C09142=1197.149,49.616,-46.613,-179.290,5.761,148.809
C09143=1197.154,49.367,-46.596,-179.293,5.760,148.810
C09144=1197.159,49.117,-46.581,-179.295,5.760,148.811
C09145=1197.164,48.868,-46.565,-179.298,5.759,148.811
C09146=1197.169,48.618,-46.548,-179.300,5.759,148.812
C09147=1197.174,48.369,-46.533,-179.303,5.758,148.812
C09148=1197.179,48.120,-46.516,-179.306,5.757,148.813
C09149=1197.184,47.870,-46.501,-179.308,5.756,148.813
C09150=1197.189,47.621,-46.484,-179.311,5.755,148.814
C09151=1197.194,47.371,-46.468,-179.313,5.755,148.815
C09152=1197.199,47.122,-46.453,-179.316,5.754,148.815
C09153=1197.204,46.872,-46.436,-179.318,5.753,148.816
C09154=1197.209,46.623,-46.421,-179.321,5.753,148.817
C09155=1197.213,46.373,-46.405,-179.323,5.752,148.817
C09156=1197.218,46.124,-46.389,-179.326,5.751,148.818
C09157=1197.223,45.874,-46.373,-179.329,5.750,148.818
C09158=1197.229,45.625,-46.357,-179.331,5.749,148.819
C09159=1197.234,45.376,-46.341,-179.334,5.749,148.820
C09160=1197.238,45.126,-46.325,-179.336,5.748,148.820
C09161=1197.244,44.877,-46.309,-179.339,5.748,148.821
C09162=1197.249,44.628,-46.293,-179.341,5.747,148.821
C09163=1197.253,44.378,-46.278,-179.344,5.746,148.822
C09164=1197.258,44.129,-46.262,-179.346,5.746,148.823
C09165=1197.263,43.879,-46.246,-179.349,5.744,148.823
C09166=1197.268,43.630,-46.230,-179.352,5.744,148.824
C09167=1197.274,43.380,-46.214,-179.354,5.743,148.824
C09168=1197.278,43.130,-46.198,-179.357,5.742,148.825
C09169=1197.284,42.881,-46.182,-179.360,5.742,148.826
C09170=1197.288,42.632,-46.167,-179.362,5.741,148.826
C09171=1197.293,42.382,-46.151,-179.364,5.740,148.827
C09172=1197.298,42.133,-46.136,-179.367,5.740,148.827
C09173=1197.304,41.883,-46.120,-179.370,5.739,148.828
C09174=1197.308,41.634,-46.103,-179.372,5.738,148.829
C09175=1197.313,41.385,-46.088,-179.374,5.738,148.829
C09176=1197.318,41.135,-46.073,-179.378,5.737,148.830
C09177=1197.323,40.885,-46.057,-179.380,5.736,148.830
C09178=1197.328,40.636,-46.041,-179.382,5.735,148.831
C09179=1197.334,40.387,-46.026,-179.385,5.735,148.832
C09180=1197.338,40.137,-46.010,-179.388,5.734,148.832
C09181=1197.343,39.888,-45.994,-179.390,5.733,148.833
C09182=1197.348,39.639,-45.978,-179.392,5.733,148.834
C09183=1197.353,39.388,-45.962,-179.395,5.732,148.834
C09184=1197.358,39.139,-45.947,-179.398,5.732,148.835
C09185=1197.363,38.890,-45.932,-179.400,5.731,148.835
C09186=1197.369,38.641,-45.916,-179.403,5.730,148.836
C09187=1197.373,38.390,-45.900,-179.406,5.729,148.837
C09188=1197.378,38.141,-45.885,-179.408,5.728,148.837
C09189=1197.383,37.892,-45.870,-179.411,5.727,148.838
C09190=1197.388,37.643,-45.853,-179.413,5.727,148.838
C09191=1197.392,37.393,-45.838,-179.416,5.726,148.839
C09192=1197.398,37.144,-45.822,-179.418,5.726,148.840
C09193=1197.403,36.895,-45.807,-179.421,5.725,148.840
C09194=1197.409,36.645,-45.791,-179.423,5.725,148.841
C09195=1197.413,36.395,-45.776,-179.426,5.724,148.842
C09196=1197.418,36.146,-45.760,-179.428,5.723,148.842
C09197=1197.423,35.897,-45.745,-179.431,5.723,148.843
C09198=1197.428,35.648,-45.730,-179.433,5.722,148.843
C09199=1197.433,35.397,-45.714,-179.436,5.722,148.844
C09200=1197.438,35.148,-45.698,-179.438,5.721,148.845
C09201=1197.443,34.899,-45.683,-179.441,5.720,148.845
C09202=1197.449,34.649,-45.668,-179.443,5.720,148.846
C09203=1197.453,34.399,-45.653,-179.447,5.718,148.847
C09204=1197.458,34.150,-45.637,-179.449,5.717,148.847
C09205=1197.463,33.900,-45.622,-179.451,5.717,148.848
C09206=1197.468,33.651,-45.607,-179.454,5.716,148.848
C09207=1197.473,33.402,-45.591,-179.457,5.716,148.849
C09208=1197.478,33.152,-45.576,-179.459,5.715,148.849
C09209=1197.483,32.903,-45.560,-179.462,5.714,148.850
C09210=1197.488,32.653,-45.545,-179.464,5.714,148.851
C09211=1197.493,32.404,-45.530,-179.467,5.713,148.851
C09212=1197.498,32.155,-45.514,-179.469,5.713,148.852
C09213=1197.503,31.904,-45.500,-179.472,5.712,148.853
C09214=1197.508,31.655,-45.484,-179.474,5.712,148.853
C09215=1197.513,31.406,-45.469,-179.477,5.711,148.854
C09216=1197.518,31.156,-45.453,-179.479,5.710,148.854
C09217=1197.523,30.907,-45.438,-179.482,5.710,148.855
C09218=1197.528,30.658,-45.423,-179.484,5.709,148.856
C09219=1197.533,30.407,-45.408,-179.487,5.709,148.856
C09220=1197.538,30.158,-45.393,-179.489,5.708,148.857
C09221=1197.543,29.909,-45.377,-179.492,5.707,148.858
C09222=1197.548,29.660,-45.362,-179.494,5.707,148.858
C09223=1197.553,29.410,-45.346,-179.497,5.706,148.859
C09224=1197.558,29.141,-45.331,-179.500,5.705,148.860
C09225=1197.564,28.872,-45.314,-179.503,5.704,148.860
C09226=1197.569,28.604,-45.298,-179.506,5.704,148.861
C09227=1197.575,28.335,-45.282,-179.508,5.703,148.862
C09228=1197.580,28.086,-45.267,-179.510,5.702,148.862
C09229=1197.584,27.836,-45.251,-179.513,5.702,148.863
C09230=1197.589,27.586,-45.236,-179.516,5.701,148.863
C09231=1197.595,27.337,-45.221,-179.518,5.701,148.864
C09232=1197.599,27.088,-45.206,-179.521,5.700,148.865
C09233=1197.605,26.838,-45.191,-179.523,5.699,148.865
C09234=1197.610,26.589,-45.176,-179.526,5.699,148.866
C09235=1197.615,26.339,-45.160,-179.528,5.698,148.867
C09236=1197.620,26.089,-45.146,-179.531,5.698,148.867
C09237=1197.625,25.840,-45.131,-179.533,5.697,148.868
C09238=1197.630,25.591,-45.116,-179.536,5.697,148.868
C09239=1197.635,25.341,-45.101,-179.539,5.696,148.869
C09240=1197.640,25.091,-45.085,-179.541,5.695,148.870
C09241=1197.645,24.842,-45.070,-179.543,5.695,148.870
C09242=1197.649,24.592,-45.056,-179.546,5.694,148.871
C09243=1197.655,24.343,-45.040,-179.549,5.694,148.872
C09244=1197.660,24.093,-45.026,-179.551,5.693,148.872
C09245=1197.665,23.844,-45.011,-179.553,5.692,148.873
C09246=1197.670,23.595,-44.996,-179.556,5.692,148.873
C09247=1197.675,23.345,-44.981,-179.559,5.691,148.874
C09248=1197.680,23.096,-44.966,-179.561,5.691,148.875
C09249=1197.685,22.846,-44.951,-179.564,5.690,148.875
C09250=1197.690,22.597,-44.936,-179.566,5.689,148.876
C09251=1197.695,22.347,-44.922,-179.569,5.689,148.877
C09252=1197.700,22.098,-44.907,-179.571,5.688,148.877
C09253=1197.705,21.848,-44.892,-179.574,5.687,148.878
C09254=1197.710,21.599,-44.877,-179.576,5.687,148.878
C09255=1197.715,21.349,-44.862,-179.579,5.686,148.879
C09256=1197.720,21.100,-44.847,-179.582,5.686,148.880
C09257=1197.726,20.850,-44.833,-179.584,5.685,148.880
C09258=1197.730,20.601,-44.818,-179.586,5.685,148.881
C09259=1197.735,20.351,-44.803,-179.589,5.684,148.882
C09260=1197.741,20.102,-44.788,-179.592,5.684,148.882
C09261=1197.746,19.852,-44.773,-179.594,5.683,148.883
C09262=1197.750,19.603,-44.758,-179.596,5.682,148.883
C09263=1197.755,19.353,-44.744,-179.599,5.682,148.884
C09264=1197.761,19.103,-44.729,-179.602,5.681,148.885
C09265=1197.766,18.854,-44.714,-179.604,5.681,148.885
C09266=1197.771,18.604,-44.700,-179.607,5.680,148.886
C09267=1197.775,18.355,-44.685,-179.609,5.679,148.887
C09268=1197.781,18.105,-44.670,-179.612,5.679,148.887
C09269=1197.786,17.856,-44.655,-179.615,5.678,148.888
C09270=1197.791,17.606,-44.641,-179.617,5.678,148.889
C09271=1197.796,17.357,-44.627,-179.619,5.677,148.889
C09272=1197.801,17.107,-44.611,-179.622,5.676,148.890
C09273=1197.806,16.857,-44.597,-179.625,5.676,148.890
C09274=1197.811,16.608,-44.582,-179.627,5.675,148.891
C09275=1197.815,16.359,-44.567,-179.630,5.675,148.892
C09276=1197.820,16.109,-44.553,-179.632,5.674,148.892
C09277=1197.826,15.859,-44.538,-179.635,5.673,148.893
C09278=1197.831,15.611,-44.524,-179.637,5.673,148.894
C09279=1197.836,15.361,-44.509,-179.640,5.672,148.894
C09280=1197.841,15.111,-44.495,-179.643,5.672,148.895
C09281=1197.846,14.861,-44.481,-179.645,5.671,148.895
C09282=1197.851,14.612,-44.466,-179.648,5.671,148.896
C09283=1197.857,14.362,-44.451,-179.650,5.671,148.897
C09284=1197.862,14.113,-44.437,-179.652,5.670,148.897
C09285=1197.866,13.863,-44.422,-179.655,5.670,148.898
C09286=1197.871,13.614,-44.407,-179.657,5.669,148.899
C09287=1197.876,13.364,-44.393,-179.660,5.669,148.899
C09288=1197.881,13.114,-44.379,-179.662,5.668,148.900
C09289=1197.887,12.865,-44.365,-179.665,5.668,148.901
C09290=1197.892,12.616,-44.349,-179.667,5.667,148.901
C09291=1197.897,12.366,-44.335,-179.670,5.666,148.902
C09292=1197.902,12.117,-44.321,-179.672,5.666,148.902
C09293=1197.907,11.867,-44.307,-179.675,5.665,148.903
C09294=1197.912,11.617,-44.292,-179.678,5.665,148.904
C09295=1197.916,11.368,-44.277,-179.680,5.664,148.904
C09296=1197.922,11.119,-44.263,-179.683,5.663,148.905
C09297=1197.927,10.869,-44.249,-179.685,5.663,148.906
C09298=1197.932,10.620,-44.235,-179.688,5.662,148.906
C09299=1197.937,10.370,-44.221,-179.691,5.662,148.907
C09300=1197.942,10.120,-44.206,-179.693,5.661,148.908
C09301=1197.946,9.871,-44.191,-179.695,5.661,148.908
C09302=1197.951,9.621,-44.177,-179.697,5.661,148.909
C09303=1197.957,9.372,-44.163,-179.700,5.660,148.910
C09304=1197.963,9.122,-44.148,-179.703,5.660,148.910
C09305=1197.968,8.873,-44.134,-179.705,5.659,148.911
C09306=1197.973,8.623,-44.120,-179.708,5.658,148.911
C09307=1197.978,8.373,-44.105,-179.710,5.658,148.912
C09308=1197.983,8.124,-44.091,-179.713,5.657,148.913
C09309=1197.988,7.874,-44.077,-179.715,5.657,148.913
C09310=1197.993,7.625,-44.063,-179.718,5.656,148.914
C09311=1197.998,7.375,-44.049,-179.720,5.656,148.915
C09312=1198.003,7.125,-44.034,-179.723,5.655,148.915
C09313=1198.008,6.876,-44.020,-179.726,5.655,148.916
C09314=1198.013,6.627,-44.006,-179.728,5.654,148.917
C09315=1198.018,6.377,-43.992,-179.730,5.654,148.917
C09316=1198.023,6.128,-43.978,-179.732,5.653,148.918
C09317=1198.028,5.878,-43.964,-179.735,5.653,148.918
C09318=1198.033,5.629,-43.950,-179.738,5.652,148.919
C09319=1198.038,5.379,-43.936,-179.740,5.652,148.920
C09320=1198.043,5.129,-43.921,-179.743,5.651,148.920
C09321=1198.048,4.880,-43.907,-179.745,5.651,148.921
C09322=1198.054,4.631,-43.893,-179.748,5.650,148.922
C09323=1198.058,4.381,-43.879,-179.751,5.650,148.922
C09324=1198.063,4.131,-43.865,-179.753,5.649,148.923
C09325=1198.068,3.882,-43.850,-179.755,5.648,148.924
C09326=1198.073,3.632,-43.836,-179.757,5.649,148.924
C09327=1198.079,3.383,-43.822,-179.760,5.648,148.925
C09328=1198.084,3.113,-43.807,-179.763,5.648,148.926
C09329=1198.090,2.844,-43.792,-179.765,5.647,148.926
C09330=1198.095,2.575,-43.777,-179.768,5.647,148.927
C09331=1198.100,2.306,-43.762,-179.771,5.645,148.928
C09332=1198.106,2.057,-43.748,-179.773,5.646,148.928
C09333=1198.110,1.807,-43.734,-179.776,5.645,148.929
C09334=1198.115,1.558,-43.720,-179.779,5.645,148.930
C09335=1198.121,1.308,-43.707,-179.781,5.644,148.930
C09336=1198.126,1.058,-43.692,-179.783,5.643,148.931
C09337=1198.131,0.809,-43.678,-179.786,5.643,148.932
C09338=1198.136,0.560,-43.664,-179.789,5.642,148.932
C09339=1198.141,0.310,-43.650,-179.791,5.642,148.933
C09340=1198.146,0.060,-43.636,-179.794,5.641,148.933
C09341=1198.151,-0.190,-43.623,-179.796,5.641,148.934
C09342=1198.156,-0.439,-43.609,-179.798,5.641,148.935
C09343=1198.161,-0.689,-43.594,-179.801,5.640,148.935
C09344=1198.166,-0.938,-43.580,-179.804,5.640,148.936
C09345=1198.171,-1.188,-43.567,-179.806,5.639,148.937
C09346=1198.176,-1.437,-43.553,-179.808,5.638,148.937
C09347=1198.181,-1.687,-43.539,-179.811,5.638,148.938
C09348=1198.187,-1.936,-43.525,-179.814,5.638,148.939
C09349=1198.192,-2.186,-43.511,-179.816,5.638,148.939
C09350=1198.196,-2.436,-43.498,-179.818,5.637,148.940
C09351=1198.202,-2.685,-43.484,-179.821,5.636,148.941
C09352=1198.207,-2.934,-43.470,-179.823,5.636,148.941
C09353=1198.213,-3.184,-43.456,-179.826,5.636,148.942
C09354=1198.217,-3.433,-43.443,-179.829,5.635,148.943
C09355=1198.222,-3.683,-43.428,-179.831,5.635,148.943
C09356=1198.228,-3.933,-43.415,-179.834,5.634,148.944
C09357=1198.233,-4.183,-43.401,-179.836,5.634,148.944
C09358=1198.237,-4.432,-43.387,-179.838,5.634,148.945
C09359=1198.243,-4.682,-43.374,-179.841,5.633,148.946
C09360=1198.248,-4.931,-43.360,-179.843,5.633,148.946
C09361=1198.253,-5.180,-43.346,-179.846,5.632,148.947
C09362=1198.258,-5.430,-43.333,-179.848,5.631,148.948
C09363=1198.263,-5.680,-43.319,-179.851,5.631,148.948
C09364=1198.268,-5.929,-43.306,-179.854,5.630,148.949
C09365=1198.273,-6.179,-43.292,-179.856,5.631,148.950
C09366=1198.278,-6.428,-43.278,-179.858,5.630,148.950
C09367=1198.284,-6.678,-43.264,-179.861,5.630,148.951
C09368=1198.288,-6.928,-43.251,-179.863,5.629,148.952
C09369=1198.294,-7.177,-43.237,-179.866,5.628,148.952
C09370=1198.298,-7.427,-43.224,-179.868,5.628,148.953
C09371=1198.304,-7.676,-43.211,-179.871,5.627,148.954
C09372=1198.309,-7.926,-43.196,-179.873,5.628,148.954
C09373=1198.313,-8.176,-43.183,-179.875,5.627,148.955
C09374=1198.319,-8.425,-43.169,-179.878,5.626,148.955
C09375=1198.324,-8.675,-43.155,-179.881,5.626,148.956
C09376=1198.329,-8.924,-43.142,-179.883,5.625,148.957
C09377=1198.334,-9.174,-43.128,-179.886,5.625,148.958
C09378=1198.339,-9.423,-43.116,-179.888,5.625,148.958
C09379=1198.344,-9.673,-43.101,-179.890,5.624,148.959
C09380=1198.350,-9.923,-43.088,-179.893,5.624,148.959
C09381=1198.354,-10.172,-43.074,-179.896,5.623,148.960
C09382=1198.359,-10.422,-43.061,-179.898,5.623,148.961
C09383=1198.364,-10.671,-43.048,-179.901,5.622,148.961
C09384=1198.369,-10.921,-43.034,-179.902,5.622,148.962
C09385=1198.375,-11.171,-43.021,-179.905,5.622,148.963
C09386=1198.379,-11.420,-43.007,-179.908,5.621,148.963
C09387=1198.385,-11.670,-42.994,-179.910,5.621,148.964
C09388=1198.390,-11.919,-42.980,-179.913,5.620,148.965
C09389=1198.395,-12.169,-42.967,-179.916,5.620,148.965
C09390=1198.400,-12.418,-42.953,-179.917,5.620,148.966
C09391=1198.405,-12.668,-42.940,-179.920,5.619,148.967
C09392=1198.410,-12.918,-42.927,-179.923,5.619,148.967
C09393=1198.416,-13.167,-42.913,-179.925,5.618,148.968
C09394=1198.420,-13.417,-42.900,-179.928,5.618,148.969
C09395=1198.426,-13.666,-42.886,-179.931,5.617,148.969
C09396=1198.430,-13.916,-42.873,-179.932,5.617,148.970
C09397=1198.436,-14.166,-42.860,-179.935,5.617,148.970
C09398=1198.440,-14.415,-42.847,-179.938,5.616,148.971
C09399=1198.446,-14.665,-42.833,-179.940,5.616,148.972
C09400=1198.451,-14.915,-42.820,-179.943,5.616,148.973
C09401=1198.456,-15.164,-42.807,-179.945,5.615,148.973
C09402=1198.461,-15.413,-42.794,-179.947,5.615,148.974
C09403=1198.467,-15.663,-42.780,-179.950,5.615,148.974
C09404=1198.472,-15.913,-42.768,-179.952,5.614,148.975
C09405=1198.477,-16.162,-42.753,-179.955,5.614,148.976
C09406=1198.482,-16.412,-42.741,-179.958,5.613,148.976
C09407=1198.487,-16.662,-42.727,-179.959,5.613,148.977
C09408=1198.492,-16.911,-42.714,-179.962,5.613,148.978
C09409=1198.497,-17.161,-42.700,-179.965,5.612,148.978
C09410=1198.502,-17.410,-42.688,-179.967,5.612,148.979
C09411=1198.507,-17.660,-42.675,-179.970,5.611,148.980
C09412=1198.512,-17.910,-42.661,-179.973,5.611,148.980
C09413=1198.517,-18.159,-42.648,-179.974,5.611,148.981
C09414=1198.523,-18.409,-42.635,-179.977,5.610,148.982
C09415=1198.528,-18.658,-42.622,-179.979,5.610,148.982
C09416=1198.534,-18.908,-42.609,-179.982,5.609,148.983
C09417=1198.538,-19.158,-42.595,-179.985,5.609,148.984
C09418=1198.543,-19.407,-42.583,-179.987,5.609,148.984
C09419=1198.548,-19.657,-42.569,-179.989,5.608,148.985
C09420=1198.553,-19.906,-42.557,-179.992,5.608,148.986
C09421=1198.559,-20.156,-42.543,-179.994,5.607,148.986
C09422=1198.564,-20.406,-42.530,-179.997,5.607,148.987
C09423=1198.569,-20.655,-42.517,-179.999,5.607,148.988
C09424=1198.574,-20.905,-42.504,179.998,5.607,148.988
C09425=1198.579,-21.154,-42.491,179.996,5.606,148.989
C09426=1198.584,-21.404,-42.478,179.993,5.605,148.989
C09427=1198.589,-21.654,-42.465,179.991,5.606,148.990
C09428=1198.594,-21.903,-42.452,179.989,5.605,148.991
C09429=1198.600,-22.153,-42.440,179.986,5.605,148.992
C09430=1198.605,-22.403,-42.426,179.984,5.604,148.992
C09431=1198.610,-22.652,-42.413,179.981,5.603,148.993
C09432=1198.615,-22.922,-42.398,179.979,5.603,148.993
C09433=1198.621,-23.191,-42.385,179.976,5.602,148.994
C09434=1198.627,-23.461,-42.371,179.974,5.603,148.995
C09435=1198.632,-23.731,-42.357,179.971,5.603,148.996
C09436=1198.637,-23.980,-42.345,179.968,5.602,148.996
C09437=1198.642,-24.230,-42.331,179.966,5.601,148.997
C09438=1198.647,-24.480,-42.318,179.963,5.601,148.998
C09439=1198.652,-24.729,-42.306,179.961,5.601,148.998
C09440=1198.657,-24.979,-42.293,179.958,5.601,148.999
C09441=1198.663,-25.229,-42.280,179.956,5.600,149.000
C09442=1198.668,-25.478,-42.267,179.954,5.599,149.000
C09443=1198.673,-25.727,-42.254,179.951,5.599,149.001
C09444=1198.678,-25.977,-42.241,179.949,5.599,149.002
C09445=1198.683,-26.227,-42.228,179.946,5.599,149.002
C09446=1198.689,-26.476,-42.216,179.944,5.598,149.003
C09447=1198.693,-26.726,-42.203,179.941,5.598,149.003
C09448=1198.698,-26.975,-42.190,179.939,5.598,149.004
C09449=1198.704,-27.225,-42.177,179.937,5.597,149.005
C09450=1198.709,-27.475,-42.164,179.934,5.597,149.005
C09451=1198.714,-27.724,-42.151,179.931,5.596,149.006
C09452=1198.719,-27.974,-42.139,179.929,5.596,149.007
C09453=1198.724,-28.223,-42.126,179.927,5.596,149.007
C09454=1198.729,-28.473,-42.113,179.924,5.596,149.008
C09455=1198.734,-28.723,-42.100,179.922,5.595,149.009
C09456=1198.739,-28.972,-42.087,179.919,5.595,149.009
C09457=1198.745,-29.222,-42.075,179.917,5.595,149.010
C09458=1198.749,-29.472,-42.062,179.914,5.594,149.011
C09459=1198.755,-29.721,-42.050,179.912,5.594,149.011
C09460=1198.760,-29.971,-42.037,179.909,5.593,149.012
C09461=1198.766,-30.220,-42.024,179.907,5.593,149.013
C09462=1198.770,-30.470,-42.011,179.905,5.593,149.013
C09463=1198.775,-30.720,-41.999,179.902,5.593,149.014
C09464=1198.781,-30.970,-41.987,179.899,5.592,149.015
C09465=1198.786,-31.219,-41.974,179.898,5.592,149.015
C09466=1198.790,-31.469,-41.961,179.895,5.592,149.016
C09467=1198.796,-31.718,-41.948,179.892,5.591,149.017
C09468=1198.801,-31.968,-41.935,179.890,5.591,149.017
C09469=1198.806,-32.217,-41.923,179.888,5.591,149.018
C09470=1198.812,-32.467,-41.911,179.885,5.591,149.019
C09471=1198.816,-32.717,-41.898,179.883,5.590,149.019
C09472=1198.821,-32.966,-41.885,179.880,5.589,149.020
C09473=1198.827,-33.216,-41.873,179.878,5.590,149.021
C09474=1198.832,-33.466,-41.861,179.876,5.589,149.021
C09475=1198.837,-33.715,-41.848,179.873,5.589,149.022
C09476=1198.842,-33.965,-41.835,179.870,5.588,149.023
C09477=1198.847,-34.214,-41.823,179.869,5.588,149.023
C09478=1198.852,-34.464,-41.811,179.866,5.588,149.024
C09479=1198.858,-34.714,-41.797,179.863,5.587,149.025
C09480=1198.863,-34.963,-41.785,179.861,5.587,149.025
C09481=1198.868,-35.214,-41.773,179.859,5.587,149.026
C09482=1198.873,-35.463,-41.760,179.856,5.586,149.026
C09483=1198.878,-35.712,-41.747,179.854,5.586,149.027
C09484=1198.883,-35.962,-41.735,179.852,5.586,149.028
C09485=1198.889,-36.212,-41.723,179.849,5.586,149.029
C09486=1198.894,-36.461,-41.710,179.846,5.585,149.029
C09487=1198.899,-36.710,-41.698,179.844,5.585,149.030
C09488=1198.904,-36.961,-41.685,179.842,5.585,149.030
C09489=1198.909,-37.210,-41.673,179.839,5.584,149.031
C09490=1198.914,-37.460,-41.661,179.837,5.584,149.032
C09491=1198.920,-37.710,-41.648,179.834,5.583,149.033
C09492=1198.925,-37.959,-41.636,179.832,5.584,149.033
C09493=1198.930,-38.209,-41.624,179.829,5.583,149.034
C09494=1198.935,-38.458,-41.611,179.827,5.582,149.034
C09495=1198.940,-38.708,-41.598,179.824,5.582,149.035
C09496=1198.945,-38.958,-41.586,179.822,5.582,149.036
C09497=1198.950,-39.207,-41.574,179.820,5.582,149.036
C09498=1198.956,-39.457,-41.562,179.817,5.581,149.037
C09499=1198.961,-39.707,-41.549,179.815,5.582,149.038
C09500=1198.966,-39.957,-41.537,179.813,5.581,149.038
C09501=1198.971,-40.206,-41.525,179.810,5.580,149.039
C09502=1198.976,-40.455,-41.513,179.807,5.580,149.040
C09503=1198.981,-40.705,-41.501,179.805,5.580,149.040
C09504=1198.986,-40.954,-41.488,179.803,5.580,149.041
C09505=1198.991,-41.205,-41.476,179.801,5.579,149.042
C09506=1198.996,-41.454,-41.464,179.798,5.579,149.042
C09507=1199.002,-41.704,-41.452,179.796,5.579,149.043
C09508=1199.007,-41.953,-41.439,179.793,5.578,149.044
C09509=1199.012,-42.203,-41.427,179.790,5.578,149.044
C09510=1199.017,-42.453,-41.415,179.788,5.578,149.045
C09511=1199.023,-42.703,-41.403,179.786,5.578,149.046
C09512=1199.027,-42.952,-41.391,179.784,5.577,149.046
C09513=1199.033,-43.202,-41.379,179.781,5.577,149.047
C09514=1199.038,-43.451,-41.366,179.779,5.577,149.048
C09515=1199.043,-43.701,-41.354,179.776,5.577,149.048
C09516=1199.049,-43.951,-41.342,179.774,5.577,149.049
C09517=1199.054,-44.200,-41.330,179.772,5.576,149.050
C09518=1199.059,-44.450,-41.318,179.769,5.576,149.050
C09519=1199.064,-44.699,-41.306,179.767,5.575,149.051
C09520=1199.069,-44.949,-41.294,179.764,5.575,149.052
C09521=1199.074,-45.198,-41.281,179.762,5.575,149.052
C09522=1199.080,-45.448,-41.270,179.760,5.574,149.053
C09523=1199.084,-45.699,-41.257,179.758,5.575,149.054
C09524=1199.090,-45.948,-41.245,179.755,5.574,149.054
C09525=1199.094,-46.198,-41.233,179.752,5.574,149.055
C09526=1199.100,-46.448,-41.222,179.750,5.574,149.056
C09527=1199.105,-46.697,-41.209,179.747,5.574,149.056
C09528=1199.110,-46.947,-41.197,179.745,5.573,149.057
C09529=1199.116,-47.197,-41.185,179.743,5.572,149.058
C09530=1199.120,-47.446,-41.173,179.741,5.573,149.058
C09531=1199.125,-47.696,-41.161,179.738,5.572,149.059
C09532=1199.131,-47.946,-41.149,179.735,5.572,149.060
C09533=1199.136,-48.195,-41.137,179.733,5.572,149.060
C09534=1199.141,-48.445,-41.125,179.731,5.571,149.061
C09535=1199.147,-48.694,-41.114,179.728,5.571,149.062
C09536=1199.152,-48.964,-41.101,179.726,5.571,149.062
C09537=1199.157,-49.235,-41.088,179.724,5.571,149.063
C09538=1199.164,-49.505,-41.075,179.721,5.570,149.064
C09539=1199.169,-49.775,-41.062,179.718,5.570,149.064
C09540=1199.174,-50.024,-41.050,179.716,5.569,149.065
C09541=1199.179,-50.274,-41.038,179.713,5.570,149.066
C09542=1199.185,-50.524,-41.026,179.711,5.569,149.066
C09543=1199.190,-50.774,-41.014,179.708,5.569,149.067
C09544=1199.194,-51.023,-41.002,179.707,5.569,149.068
C09545=1199.200,-51.273,-40.990,179.704,5.568,149.068
C09546=1199.205,-51.523,-40.978,179.701,5.568,149.069
C09547=1199.210,-51.772,-40.967,179.699,5.568,149.070
C09548=1199.215,-52.022,-40.955,179.696,5.568,149.070
C09549=1199.221,-52.271,-40.943,179.694,5.567,149.071
C09550=1199.226,-52.520,-40.932,179.692,5.567,149.072
C09551=1199.231,-52.770,-40.920,179.690,5.567,149.072
C09552=1199.237,-53.020,-40.908,179.687,5.566,149.073
C09553=1199.241,-53.270,-40.897,179.685,5.567,149.074
C09554=1199.246,-53.519,-40.884,179.682,5.566,149.074
C09555=1199.252,-53.769,-40.872,179.680,5.566,149.075
C09556=1199.257,-54.019,-40.861,179.678,5.566,149.076
C09557=1199.262,-54.269,-40.849,179.675,5.565,149.076
C09558=1199.267,-54.519,-40.837,179.673,5.565,149.077
C09559=1199.272,-54.768,-40.826,179.670,5.565,149.078
C09560=1199.278,-55.018,-40.814,179.668,5.565,149.078
C09561=1199.282,-55.267,-40.802,179.666,5.564,149.079
C09562=1199.288,-55.516,-40.790,179.664,5.564,149.080
C09563=1199.293,-55.766,-40.779,179.661,5.564,149.080
C09564=1199.298,-56.016,-40.767,179.658,5.564,149.081
C09565=1199.303,-56.266,-40.755,179.656,5.564,149.082
C09566=1199.308,-56.516,-40.744,179.654,5.563,149.082
C09567=1199.314,-56.766,-40.732,179.651,5.563,149.083
C09568=1199.318,-57.015,-40.721,179.649,5.563,149.084
C09569=1199.324,-57.264,-40.709,179.647,5.563,149.084
C09570=1199.330,-57.514,-40.698,179.644,5.562,149.085
C09571=1199.334,-57.764,-40.686,179.642,5.562,149.086
C09572=1199.340,-58.014,-40.674,179.640,5.562,149.086
C09573=1199.345,-58.264,-40.663,179.637,5.561,149.087
C09574=1199.350,-58.513,-40.651,179.635,5.562,149.088
C09575=1199.355,-58.763,-40.640,179.632,5.561,149.088
C09576=1199.361,-59.012,-40.628,179.630,5.560,149.089
C09577=1199.365,-59.262,-40.617,179.628,5.561,149.090
C09578=1199.371,-59.512,-40.605,179.625,5.560,149.090
C09579=1199.376,-59.762,-40.594,179.623,5.561,149.091
C09580=1199.381,-60.011,-40.582,179.620,5.560,149.092
C09581=1199.386,-60.261,-40.570,179.618,5.559,149.092
C09582=1199.392,-60.510,-40.559,179.616,5.560,149.093
C09583=1199.397,-60.760,-40.547,179.614,5.559,149.094
C09584=1199.402,-61.010,-40.536,179.611,5.559,149.094
C09585=1199.407,-61.260,-40.524,179.609,5.559,149.095
C09586=1199.412,-61.509,-40.513,179.607,5.558,149.095
C09587=1199.417,-61.758,-40.502,179.604,5.558,149.096
C09588=1199.423,-62.008,-40.490,179.602,5.558,149.097
C09589=1199.427,-62.258,-40.479,179.599,5.558,149.098
C09590=1199.433,-62.508,-40.467,179.597,5.557,149.098
C09591=1199.437,-62.758,-40.456,179.595,5.557,149.099
C09592=1199.444,-63.007,-40.445,179.592,5.557,149.099
C09593=1199.448,-63.257,-40.433,179.590,5.557,149.100
C09594=1199.454,-63.507,-40.422,179.588,5.557,149.101
C09595=1199.459,-63.757,-40.410,179.585,5.556,149.102
C09596=1199.464,-64.006,-40.398,179.583,5.556,149.102
C09597=1199.469,-64.255,-40.387,179.581,5.556,149.103
C09598=1199.474,-64.505,-40.376,179.578,5.555,149.103
C09599=1199.480,-64.756,-40.365,179.576,5.556,149.104
C09600=1199.484,-65.005,-40.354,179.573,5.555,149.105
C09601=1199.490,-65.254,-40.342,179.572,5.555,149.105
C09602=1199.495,-65.504,-40.331,179.569,5.555,149.106
C09603=1199.501,-65.754,-40.319,179.566,5.555,149.107
C09604=1199.505,-66.004,-40.308,179.564,5.555,149.107
C09605=1199.511,-66.253,-40.298,179.561,5.554,149.108
C09606=1199.516,-66.503,-40.286,179.559,5.554,149.109
C09607=1199.521,-66.753,-40.274,179.557,5.554,149.109
C09608=1199.526,-67.002,-40.263,179.555,5.554,149.110
C09609=1199.532,-67.252,-40.252,179.552,5.554,149.111
C09610=1199.537,-67.502,-40.241,179.550,5.554,149.111
C09611=1199.542,-67.752,-40.229,179.548,5.553,149.112
C09612=1199.547,-68.001,-40.218,179.546,5.553,149.113
C09613=1199.552,-68.251,-40.208,179.543,5.553,149.113
C09614=1199.558,-68.501,-40.196,179.540,5.552,149.114
C09615=1199.563,-68.750,-40.185,179.538,5.553,149.115
C09616=1199.568,-68.999,-40.173,179.536,5.552,149.115
C09617=1199.574,-69.250,-40.162,179.534,5.552,149.116
C09618=1199.578,-69.500,-40.151,179.531,5.552,149.117
C09619=1199.584,-69.749,-40.140,179.528,5.551,149.117
C09620=1199.589,-69.999,-40.129,179.527,5.551,149.118
C09621=1199.594,-70.249,-40.118,179.524,5.551,149.119
C09622=1199.599,-70.498,-40.107,179.522,5.551,149.119
C09623=1199.605,-70.748,-40.096,179.519,5.551,149.120
C09624=1199.610,-70.998,-40.084,179.517,5.550,149.121
C09625=1199.615,-71.247,-40.073,179.515,5.550,149.121
C09626=1199.620,-71.497,-40.063,179.513,5.550,149.122
C09627=1199.625,-71.747,-40.051,179.510,5.549,149.123
C09628=1199.631,-71.996,-40.040,179.508,5.550,149.123
C09629=1199.636,-72.246,-40.029,179.505,5.549,149.124
C09630=1199.641,-72.496,-40.018,179.504,5.549,149.124
C09631=1199.647,-72.746,-40.007,179.501,5.549,149.125
C09632=1199.651,-72.995,-39.996,179.498,5.548,149.126
C09633=1199.657,-73.244,-39.985,179.496,5.549,149.127
C09634=1199.662,-73.495,-39.974,179.494,5.548,149.127
C09635=1199.667,-73.744,-39.963,179.492,5.548,149.128
C09636=1199.673,-73.994,-39.952,179.489,5.548,149.128
C09637=1199.677,-74.243,-39.941,179.486,5.548,149.129
C09638=1199.683,-74.494,-39.930,179.484,5.548,149.130
C09639=1199.689,-74.743,-39.919,179.482,5.547,149.130
C09640=1199.694,-75.014,-39.907,179.480,5.547,149.131
C09641=1199.700,-75.284,-39.895,179.477,5.547,149.132
C09642=1199.705,-75.555,-39.883,179.475,5.547,149.132
C09643=1199.711,-75.827,-39.872,179.472,5.546,149.133
C09644=1199.716,-76.075,-39.861,179.470,5.547,149.134
C09645=1199.721,-76.325,-39.849,179.467,5.546,149.135
C09646=1199.727,-76.575,-39.839,179.465,5.546,149.135
C09647=1199.732,-76.825,-39.829,179.463,5.546,149.136
C09648=1199.737,-77.075,-39.817,179.460,5.545,149.136
C09649=1199.743,-77.324,-39.807,179.458,5.546,149.137
C09650=1199.747,-77.574,-39.795,179.456,5.545,149.138
C09651=1199.753,-77.823,-39.785,179.454,5.546,149.139
C09652=1199.758,-78.073,-39.774,179.451,5.545,149.139
C09653=1199.763,-78.323,-39.763,179.449,5.544,149.140
C09654=1199.769,-78.573,-39.752,179.447,5.545,149.141
C09655=1199.774,-78.823,-39.741,179.444,5.544,149.141
C09656=1199.779,-79.072,-39.730,179.442,5.544,149.142
C09657=1199.784,-79.322,-39.720,179.440,5.544,149.142
C09658=1199.790,-79.572,-39.709,179.438,5.544,149.143
C09659=1199.794,-79.821,-39.698,179.435,5.544,149.144
C09660=1199.800,-80.071,-39.688,179.433,5.543,149.144
C09661=1199.805,-80.320,-39.677,179.431,5.543,149.145
C09662=1199.810,-80.571,-39.665,179.428,5.543,149.146
C09663=1199.816,-80.820,-39.655,179.426,5.543,149.146
C09664=1199.821,-81.070,-39.644,179.424,5.542,149.147
C09665=1199.826,-81.320,-39.634,179.421,5.542,149.148
C09666=1199.831,-81.569,-39.622,179.419,5.542,149.148
C09667=1199.837,-81.819,-39.612,179.416,5.542,149.149
C09668=1199.842,-82.069,-39.602,179.414,5.542,149.150
C09669=1199.847,-82.318,-39.591,179.412,5.542,149.150
C09670=1199.852,-82.568,-39.580,179.410,5.542,149.151
C09671=1199.857,-82.818,-39.570,179.407,5.542,149.152
C09672=1199.862,-83.067,-39.559,179.405,5.541,149.152
C09673=1199.868,-83.317,-39.548,179.403,5.541,149.153
C09674=1199.873,-83.567,-39.538,179.400,5.541,149.154
C09675=1199.878,-83.817,-39.528,179.398,5.541,149.154
C09676=1199.883,-84.066,-39.516,179.396,5.541,149.155
C09677=1199.889,-84.316,-39.506,179.394,5.541,149.155
C09678=1199.894,-84.566,-39.496,179.391,5.540,149.156
C09679=1199.899,-84.815,-39.485,179.389,5.541,149.157
C09680=1199.904,-85.065,-39.474,179.387,5.540,149.158
C09681=1199.909,-85.315,-39.464,179.384,5.539,149.158
C09682=1199.914,-85.565,-39.453,179.382,5.540,149.159
C09683=1199.920,-85.814,-39.442,179.380,5.539,149.159
C09684=1199.925,-86.064,-39.432,179.378,5.540,149.160
C09685=1199.930,-86.314,-39.422,179.375,5.539,149.161
C09686=1199.935,-86.564,-39.411,179.373,5.539,149.161
C09687=1199.941,-86.813,-39.400,179.371,5.539,149.162
C09688=1199.946,-87.063,-39.390,179.368,5.538,149.163
C09689=1199.951,-87.313,-39.379,179.366,5.538,149.163
C09690=1199.957,-87.562,-39.369,179.364,5.538,149.164
C09691=1199.962,-87.813,-39.359,179.362,5.538,149.165
C09692=1199.967,-88.061,-39.348,179.359,5.538,149.165
C09693=1199.972,-88.312,-39.337,179.357,5.538,149.166
C09694=1199.978,-88.561,-39.327,179.355,5.538,149.167
C09695=1199.983,-88.811,-39.316,179.353,5.538,149.167
C09696=1199.988,-89.061,-39.306,179.350,5.537,149.168
C09697=1199.994,-89.311,-39.296,179.348,5.537,149.169
C09698=1199.999,-89.560,-39.285,179.346,5.537,149.169
C09699=1200.004,-89.810,-39.274,179.343,5.537,149.170
C09700=1200.009,-90.060,-39.264,179.341,5.537,149.170
C09701=1200.015,-90.310,-39.254,179.339,5.536,149.171
C09702=1200.019,-90.559,-39.244,179.337,5.537,149.172
C09703=1200.025,-90.809,-39.233,179.334,5.536,149.173
C09704=1200.030,-91.059,-39.223,179.332,5.536,149.173
C09705=1200.035,-91.309,-39.213,179.330,5.536,149.174
C09706=1200.041,-91.558,-39.202,179.327,5.535,149.174
C09707=1200.046,-91.809,-39.192,179.325,5.536,149.175
C09708=1200.051,-92.057,-39.181,179.323,5.535,149.176
C09709=1200.057,-92.307,-39.171,179.321,5.535,149.176
C09710=1200.061,-92.557,-39.161,179.318,5.535,149.177
C09711=1200.067,-92.807,-39.151,179.316,5.535,149.178
C09712=1200.072,-93.056,-39.140,179.314,5.534,149.178
C09713=1200.077,-93.306,-39.130,179.312,5.535,149.179
C09714=1200.083,-93.556,-39.120,179.309,5.534,149.180
C09715=1200.088,-93.806,-39.109,179.307,5.534,149.180
C09716=1200.093,-94.056,-39.099,179.305,5.534,149.181
C09717=1200.098,-94.305,-39.089,179.303,5.534,149.182
C09718=1200.103,-94.555,-39.079,179.300,5.534,149.182
C09719=1200.109,-94.805,-39.068,179.298,5.533,149.183
C09720=1200.114,-95.054,-39.058,179.296,5.534,149.184
C09721=1200.119,-95.304,-39.048,179.293,5.533,149.184
C09722=1200.124,-95.554,-39.038,179.291,5.533,149.185
C09723=1200.130,-95.803,-39.028,179.289,5.533,149.185
C09724=1200.135,-96.053,-39.017,179.287,5.533,149.186
C09725=1200.141,-96.303,-39.007,179.284,5.533,149.187
C09726=1200.146,-96.553,-38.997,179.282,5.533,149.187
C09727=1200.150,-96.802,-38.987,179.280,5.532,149.188
C09728=1200.156,-97.052,-38.977,179.277,5.533,149.189
C09729=1200.162,-97.302,-38.967,179.275,5.532,149.189
C09730=1200.167,-97.552,-38.957,179.273,5.532,149.190
C09731=1200.172,-97.802,-38.946,179.271,5.532,149.191
C09732=1200.177,-98.051,-38.937,179.268,5.532,149.191
C09733=1200.183,-98.301,-38.926,179.266,5.531,149.192
C09734=1200.188,-98.551,-38.916,179.264,5.531,149.193
C09735=1200.194,-98.801,-38.906,179.261,5.531,149.193
C09736=1200.198,-99.050,-38.896,179.259,5.531,149.194
C09737=1200.203,-99.300,-38.886,179.257,5.531,149.194
C09738=1200.209,-99.550,-38.875,179.255,5.531,149.195
C09739=1200.214,-99.799,-38.866,179.252,5.531,149.196
C09740=1200.219,-100.050,-38.856,179.250,5.530,149.196
C09741=1200.225,-100.299,-38.846,179.248,5.531,149.197
C09742=1200.230,-100.549,-38.835,179.246,5.530,149.198
C09743=1200.235,-100.798,-38.826,179.244,5.530,149.198
C09744=1200.241,-101.070,-38.814,179.241,5.530,149.199
C09745=1200.247,-101.342,-38.804,179.239,5.529,149.200
C09746=1200.252,-101.613,-38.793,179.236,5.530,149.200
C09747=1200.258,-101.884,-38.782,179.234,5.529,149.201
C09748=1200.263,-102.134,-38.773,179.232,5.530,149.202
C09749=1200.269,-102.384,-38.762,179.229,5.529,149.203
C09750=1200.274,-102.633,-38.752,179.227,5.529,149.203
C09751=1200.279,-102.883,-38.743,179.225,5.529,149.204
C09752=1200.284,-103.133,-38.732,179.223,5.529,149.204
C09753=1200.290,-103.383,-38.723,179.220,5.528,149.205
C09754=1200.295,-103.632,-38.713,179.218,5.528,149.206
C09755=1200.300,-103.882,-38.703,179.216,5.528,149.206
C09756=1200.305,-104.132,-38.692,179.214,5.528,149.207
C09757=1200.310,-104.382,-38.683,179.211,5.528,149.208
C09758=1200.316,-104.631,-38.673,179.209,5.528,149.208
C09759=1200.322,-104.881,-38.663,179.207,5.528,149.209
C09760=1200.327,-105.130,-38.653,179.204,5.527,149.210
C09761=1200.332,-105.381,-38.643,179.202,5.528,149.210
C09762=1200.337,-105.630,-38.634,179.200,5.527,149.211
C09763=1200.342,-105.880,-38.624,179.198,5.527,149.211
C09764=1200.348,-106.130,-38.614,179.195,5.527,149.212
C09765=1200.353,-106.379,-38.604,179.193,5.527,149.213
C09766=1200.358,-106.629,-38.594,179.191,5.526,149.213
C09767=1200.363,-106.879,-38.585,179.189,5.527,149.214
C09768=1200.369,-107.129,-38.575,179.186,5.526,149.215
C09769=1200.374,-107.378,-38.565,179.185,5.526,149.215
C09770=1200.380,-107.628,-38.556,179.182,5.526,149.216
C09771=1200.385,-107.878,-38.545,179.180,5.526,149.217
C09772=1200.389,-108.128,-38.535,179.178,5.526,149.217
C09773=1200.395,-108.378,-38.526,179.176,5.526,149.218
C09774=1200.400,-108.627,-38.516,179.173,5.526,149.219
C09775=1200.406,-108.877,-38.506,179.171,5.526,149.219
C09776=1200.411,-109.126,-38.497,179.169,5.525,149.220
C09777=1200.416,-109.377,-38.487,179.167,5.526,149.221
C09778=1200.421,-109.627,-38.478,179.165,5.525,149.221
C09779=1200.427,-109.876,-38.468,179.162,5.525,149.222
C09780=1200.432,-110.125,-38.458,179.160,5.525,149.222
C09781=1200.438,-110.376,-38.448,179.158,5.525,149.223
C09782=1200.443,-110.625,-38.438,179.155,5.524,149.224
C09783=1200.448,-110.876,-38.429,179.153,5.525,149.224
C09784=1200.453,-111.125,-38.419,179.151,5.524,149.225
C09785=1200.458,-111.375,-38.410,179.149,5.524,149.226
C09786=1200.464,-111.625,-38.400,179.146,5.524,149.226
C09787=1200.469,-111.874,-38.391,179.145,5.524,149.227
C09788=1200.475,-112.124,-38.381,179.142,5.524,149.227
C09789=1200.480,-112.373,-38.371,179.140,5.524,149.228
C09790=1200.485,-112.623,-38.362,179.138,5.523,149.229
C09791=1200.490,-112.873,-38.351,179.136,5.524,149.229
C09792=1200.495,-113.123,-38.343,179.133,5.523,149.230
C09793=1200.501,-113.373,-38.332,179.132,5.523,149.231
C09794=1200.506,-113.623,-38.323,179.129,5.523,149.231
C09795=1200.511,-113.872,-38.313,179.127,5.523,149.232
C09796=1200.517,-114.122,-38.304,179.125,5.522,149.232
C09797=1200.522,-114.371,-38.294,179.122,5.523,149.233
C09798=1200.527,-114.621,-38.285,179.120,5.522,149.234
C09799=1200.533,-114.871,-38.276,179.118,5.522,149.234
C09800=1200.538,-115.121,-38.266,179.116,5.522,149.235
C09801=1200.543,-115.371,-38.257,179.114,5.522,149.236
C09802=1200.548,-115.621,-38.247,179.112,5.522,149.236
C09803=1200.553,-115.871,-38.238,179.109,5.522,149.237
C09804=1200.559,-116.120,-38.228,179.108,5.522,149.238
C09805=1200.564,-116.370,-38.219,179.105,5.522,149.238
C09806=1200.570,-116.620,-38.208,179.103,5.522,149.239
C09807=1200.575,-116.869,-38.200,179.101,5.521,149.239
C09808=1200.580,-117.119,-38.191,179.099,5.522,149.240
C09809=1200.586,-117.369,-38.180,179.096,5.521,149.241
C09810=1200.591,-117.619,-38.172,179.094,5.521,149.241
C09811=1200.596,-117.869,-38.163,179.092,5.521,149.242
C09812=1200.602,-118.118,-38.152,179.089,5.521,149.243
C09813=1200.607,-118.368,-38.144,179.087,5.520,149.243
C09814=1200.612,-118.617,-38.133,179.085,5.521,149.244
C09815=1200.618,-118.867,-38.124,179.083,5.520,149.244
C09816=1200.623,-119.117,-38.116,179.081,5.520,149.245
C09817=1200.628,-119.367,-38.105,179.078,5.520,149.246
C09818=1200.633,-119.617,-38.096,179.077,5.520,149.246
C09819=1200.639,-119.866,-38.088,179.074,5.520,149.247
C09820=1200.644,-120.116,-38.077,179.072,5.520,149.248
C09821=1200.649,-120.366,-38.068,179.070,5.519,149.248
C09822=1200.655,-120.616,-38.060,179.068,5.520,149.249
C09823=1200.660,-120.865,-38.049,179.065,5.519,149.250
C09824=1200.665,-121.115,-38.040,179.063,5.519,149.250
C09825=1200.670,-121.366,-38.031,179.061,5.519,149.251
C09826=1200.675,-121.615,-38.022,179.059,5.519,149.251
C09827=1200.681,-121.865,-38.012,179.057,5.519,149.252
C09828=1200.686,-122.115,-38.003,179.054,5.519,149.253
C09829=1200.691,-122.365,-37.994,179.053,5.519,149.253
C09830=1200.697,-122.614,-37.984,179.050,5.519,149.254
C09831=1200.702,-122.863,-37.976,179.048,5.519,149.255
C09832=1200.708,-123.113,-37.967,179.046,5.518,149.255
C09833=1200.713,-123.363,-37.958,179.044,5.519,149.256
C09834=1200.718,-123.613,-37.948,179.041,5.518,149.256
C09835=1200.723,-123.863,-37.939,179.039,5.518,149.257
C09836=1200.729,-124.112,-37.930,179.037,5.517,149.258
C09837=1200.734,-124.362,-37.921,179.035,5.518,149.258
C09838=1200.740,-124.612,-37.911,179.032,5.517,149.259
C09839=1200.745,-124.862,-37.902,179.031,5.517,149.260
C09840=1200.750,-125.111,-37.893,179.028,5.517,149.260
C09841=1200.755,-125.361,-37.884,179.026,5.517,149.261
C09842=1200.761,-125.611,-37.874,179.024,5.517,149.261
C09843=1200.766,-125.861,-37.866,179.022,5.517,149.262
C09844=1200.771,-126.111,-37.856,179.020,5.517,149.263
C09845=1200.776,-126.360,-37.847,179.017,5.517,149.263
C09846=1200.782,-126.611,-37.838,179.016,5.517,149.264
C09847=1200.787,-126.860,-37.829,179.013,5.516,149.265
C09848=1200.366,-126.871,-37.867,179.009,5.519,149.266
C09849=1200.361,-126.622,-37.876,179.011,5.520,149.266
C09850=1200.355,-126.371,-37.886,179.013,5.520,149.265
C09851=1200.350,-126.122,-37.895,179.016,5.521,149.265
C09852=1200.344,-125.872,-37.904,179.018,5.520,149.264
C09853=1200.339,-125.622,-37.912,179.020,5.521,149.263
C09854=1200.334,-125.373,-37.922,179.022,5.521,149.263
C09855=1200.328,-125.122,-37.932,179.025,5.521,149.262
C09856=1200.323,-124.873,-37.940,179.026,5.521,149.262
C09857=1200.318,-124.623,-37.949,179.028,5.521,149.261
C09858=1200.312,-124.374,-37.958,179.031,5.521,149.260
C09859=1200.307,-124.124,-37.968,179.033,5.521,149.260
C09860=1200.302,-123.874,-37.977,179.035,5.521,149.259
C09861=1200.296,-123.624,-37.986,179.037,5.521,149.259
C09862=1200.291,-123.374,-37.995,179.040,5.522,149.258
C09863=1200.285,-123.124,-38.004,179.042,5.521,149.257
C09864=1200.280,-122.875,-38.014,179.044,5.522,149.257
C09865=1200.275,-122.625,-38.023,179.046,5.522,149.256
C09866=1200.270,-122.375,-38.032,179.049,5.522,149.255
C09867=1200.264,-122.125,-38.041,179.050,5.522,149.255
C09868=1200.259,-121.876,-38.051,179.053,5.523,149.254
C09869=1200.254,-121.626,-38.060,179.055,5.522,149.254
C09870=1200.248,-121.376,-38.069,179.057,5.523,149.253
C09871=1200.243,-121.127,-38.079,179.059,5.522,149.252
C09872=1200.238,-120.877,-38.088,179.062,5.523,149.252
C09873=1200.232,-120.627,-38.097,179.064,5.523,149.251
C09874=1200.227,-120.377,-38.106,179.065,5.523,149.250
C09875=1200.222,-120.128,-38.116,179.068,5.523,149.250
C09876=1200.216,-119.877,-38.125,179.070,5.523,149.249
C09877=1200.211,-119.628,-38.134,179.072,5.524,149.248
C09878=1200.206,-119.378,-38.144,179.074,5.523,149.248
C09879=1200.201,-119.128,-38.153,179.077,5.524,149.247
C09880=1200.195,-118.878,-38.162,179.079,5.524,149.247
C09881=1200.191,-118.628,-38.172,179.081,5.524,149.246
C09882=1200.185,-118.378,-38.182,179.083,5.524,149.245
C09883=1200.180,-118.129,-38.191,179.086,5.524,149.245
C09884=1200.175,-117.879,-38.200,179.088,5.524,149.244
C09885=1200.169,-117.629,-38.210,179.090,5.525,149.243
C09886=1200.164,-117.380,-38.219,179.092,5.524,149.243
C09887=1200.159,-117.130,-38.228,179.095,5.525,149.242
C09888=1200.153,-116.880,-38.238,179.096,5.525,149.242
C09889=1200.148,-116.631,-38.247,179.099,5.525,149.241
C09890=1200.143,-116.380,-38.257,179.101,5.525,149.240
C09891=1200.138,-116.131,-38.266,179.103,5.526,149.240
C09892=1200.133,-115.881,-38.275,179.105,5.525,149.239
C09893=1200.127,-115.632,-38.285,179.107,5.526,149.238
C09894=1200.122,-115.382,-38.294,179.110,5.526,149.238
C09895=1200.116,-115.132,-38.304,179.112,5.526,149.237
C09896=1200.111,-114.883,-38.313,179.114,5.526,149.236
C09897=1200.105,-114.632,-38.323,179.116,5.526,149.236
C09898=1200.101,-114.382,-38.333,179.119,5.526,149.235
C09899=1200.096,-114.133,-38.342,179.121,5.527,149.235
C09900=1200.090,-113.883,-38.352,179.123,5.526,149.234
C09901=1200.085,-113.633,-38.361,179.125,5.526,149.233
C09902=1200.079,-113.384,-38.371,179.127,5.527,149.233
C09903=1200.074,-113.134,-38.380,179.129,5.526,149.232
C09904=1200.069,-112.884,-38.390,179.132,5.527,149.231
C09905=1200.063,-112.634,-38.399,179.133,5.527,149.231
C09906=1200.058,-112.385,-38.409,179.136,5.527,149.230
C09907=1200.053,-112.135,-38.418,179.138,5.527,149.229
C09908=1200.048,-111.885,-38.429,179.140,5.528,149.229
C09909=1200.042,-111.635,-38.438,179.143,5.527,149.228
C09910=1200.037,-111.385,-38.448,179.145,5.528,149.228
C09911=1200.032,-111.136,-38.457,179.147,5.528,149.227
C09912=1200.026,-110.886,-38.467,179.149,5.528,149.226
C09913=1200.021,-110.636,-38.476,179.151,5.528,149.226
C09914=1200.015,-110.387,-38.486,179.154,5.528,149.225
C09915=1200.011,-110.137,-38.496,179.156,5.528,149.224
C09916=1200.005,-109.886,-38.506,179.158,5.529,149.224
C09917=1200.000,-109.637,-38.515,179.160,5.528,149.223
C09918=1199.994,-109.387,-38.525,179.163,5.529,149.222
C09919=1199.990,-109.138,-38.534,179.164,5.529,149.222
C09920=1199.984,-108.888,-38.545,179.167,5.529,149.221
C09921=1199.979,-108.638,-38.553,179.169,5.529,149.220
C09922=1199.974,-108.388,-38.564,179.171,5.530,149.220
C09923=1199.969,-108.138,-38.573,179.173,5.529,149.219
C09924=1199.963,-107.889,-38.583,179.176,5.530,149.219
C09925=1199.957,-107.639,-38.593,179.178,5.530,149.218
C09926=1199.952,-107.389,-38.602,179.180,5.530,149.217
C09927=1199.947,-107.139,-38.613,179.182,5.530,149.217
C09928=1199.942,-106.890,-38.622,179.185,5.530,149.216
C09929=1199.936,-106.640,-38.632,179.187,5.530,149.215
C09930=1199.932,-106.391,-38.642,179.189,5.530,149.215
C09931=1199.926,-106.141,-38.652,179.192,5.530,149.214
C09932=1199.921,-105.890,-38.662,179.194,5.531,149.214
C09933=1199.916,-105.641,-38.671,179.196,5.531,149.213
C09934=1199.910,-105.391,-38.681,179.198,5.531,149.212
C09935=1199.905,-105.142,-38.691,179.201,5.532,149.212
C09936=1199.899,-104.892,-38.701,179.203,5.531,149.211
C09937=1199.894,-104.642,-38.711,179.205,5.532,149.210
C09938=1199.890,-104.393,-38.721,179.207,5.532,149.210
C09939=1199.884,-104.142,-38.730,179.210,5.532,149.209
C09940=1199.879,-103.893,-38.740,179.212,5.532,149.208
C09941=1199.873,-103.644,-38.750,179.214,5.532,149.208
C09942=1199.868,-103.393,-38.761,179.216,5.532,149.207
C09943=1199.863,-103.143,-38.769,179.219,5.532,149.206
C09944=1199.858,-102.894,-38.780,179.220,5.532,149.206
C09945=1199.852,-102.644,-38.790,179.223,5.533,149.205
C09946=1199.848,-102.394,-38.800,179.225,5.532,149.204
C09947=1199.842,-102.145,-38.810,179.228,5.533,149.204
C09948=1199.836,-101.895,-38.820,179.229,5.533,149.203
C09949=1199.831,-101.623,-38.831,179.232,5.533,149.203
C09950=1199.826,-101.352,-38.841,179.235,5.534,149.202
C09951=1199.819,-101.081,-38.852,179.237,5.533,149.201
C09952=1199.814,-100.809,-38.863,179.239,5.534,149.200
C09953=1199.808,-100.560,-38.873,179.242,5.533,149.200
C09954=1199.803,-100.310,-38.884,179.244,5.534,149.199
C09955=1199.798,-100.060,-38.893,179.246,5.534,149.198
C09956=1199.793,-99.811,-38.903,179.249,5.534,149.198
C09957=1199.787,-99.560,-38.913,179.250,5.534,149.197
C09958=1199.783,-99.311,-38.923,179.253,5.535,149.197
C09959=1199.777,-99.061,-38.933,179.255,5.535,149.196
C09960=1199.771,-98.812,-38.943,179.258,5.535,149.195
C09961=1199.766,-98.561,-38.954,179.260,5.535,149.195
C09962=1199.761,-98.312,-38.964,179.262,5.535,149.194
C09963=1199.756,-98.063,-38.974,179.265,5.535,149.193
C09964=1199.751,-97.812,-38.984,179.266,5.535,149.193
C09965=1199.745,-97.562,-38.994,179.269,5.536,149.192
C09966=1199.740,-97.313,-39.003,179.271,5.535,149.191
C09967=1199.735,-97.063,-39.014,179.274,5.536,149.191
C09968=1199.730,-96.813,-39.024,179.275,5.536,149.190
C09969=1199.724,-96.564,-39.034,179.278,5.536,149.189
C09970=1199.718,-96.314,-39.045,179.280,5.536,149.189
C09971=1199.714,-96.064,-39.055,179.282,5.537,149.188
C09972=1199.708,-95.815,-39.065,179.284,5.536,149.188
C09973=1199.703,-95.565,-39.075,179.287,5.537,149.187
C09974=1199.698,-95.315,-39.086,179.289,5.536,149.186
C09975=1199.692,-95.065,-39.096,179.291,5.537,149.186
C09976=1199.687,-94.816,-39.105,179.294,5.538,149.185
C09977=1199.682,-94.566,-39.116,179.296,5.537,149.184
C09978=1199.677,-94.316,-39.126,179.298,5.538,149.184
C09979=1199.672,-94.066,-39.137,179.300,5.538,149.183
C09980=1199.666,-93.816,-39.147,179.303,5.538,149.182
C09981=1199.661,-93.567,-39.157,179.305,5.538,149.182
C09982=1199.656,-93.317,-39.167,179.307,5.538,149.181
C09983=1199.651,-93.067,-39.177,179.309,5.538,149.180
C09984=1199.645,-92.818,-39.188,179.312,5.538,149.180
C09985=1199.640,-92.568,-39.198,179.313,5.538,149.179
C09986=1199.635,-92.318,-39.208,179.316,5.539,149.178
C09987=1199.629,-92.069,-39.219,179.319,5.539,149.178
C09988=1199.625,-91.819,-39.229,179.321,5.539,149.177
C09989=1199.619,-91.569,-39.239,179.323,5.540,149.177
C09990=1199.614,-91.319,-39.249,179.325,5.539,149.176
C09991=1199.609,-91.069,-39.260,179.328,5.540,149.175
C09992=1199.603,-90.820,-39.270,179.330,5.539,149.174
C09993=1199.598,-90.570,-39.281,179.332,5.540,149.174
C09994=1199.593,-90.321,-39.291,179.334,5.540,149.173
C09995=1199.588,-90.070,-39.302,179.337,5.540,149.173
C09996=1199.582,-89.821,-39.312,179.338,5.540,149.172
//INST
///DATE 2021/06/15 17:24
///ATTR SC,RW,RJ
////FRAME ROBOT
///GROUP1 RB1
NOP
MOVL C00000 V=800.0 PL=0
MOVL C00001 V=800.0 PL=0
MOVL C00002 V=800.0 PL=0
MOVL C00003 V=800.0 PL=0
MOVL C00004 V=800.0 PL=0
MOVL C00005 V=800.0 PL=0
MOVL C00006 V=800.0 PL=0
MOVL C00007 V=800.0 PL=0
MOVL C00008 V=800.0 PL=0
MOVL C00009 V=800.0 PL=0
MOVL C00010 V=800.0 PL=0
MOVL C00011 V=800.0 PL=0
MOVL C00012 V=800.0 PL=0
MOVL C00013 V=800.0 PL=0
MOVL C00014 V=800.0 PL=0
MOVL C00015 V=800.0 PL=0
MOVL C00016 V=800.0 PL=0
MOVL C00017 V=800.0 PL=0
MOVL C00018 V=800.0 PL=0
MOVL C00019 V=800.0 PL=0
MOVL C00020 V=800.0 PL=0
MOVL C00021 V=800.0 PL=0
MOVL C00022 V=800.0 PL=0
MOVL C00023 V=800.0 PL=0
MOVL C00024 V=800.0 PL=0
MOVL C00025 V=800.0 PL=0
MOVL C00026 V=800.0 PL=0
MOVL C00027 V=800.0 PL=0
MOVL C00028 V=800.0 PL=0
MOVL C00029 V=800.0 PL=0
MOVL C00030 V=800.0 PL=0
MOVL C00031 V=800.0 PL=0
MOVL C00032 V=800.0 PL=0
MOVL C00033 V=800.0 PL=0
MOVL C00034 V=800.0 PL=0
MOVL C00035 V=800.0 PL=0
MOVL C00036 V=800.0 PL=0
MOVL C00037 V=800.0 PL=0
MOVL C00038 V=800.0 PL=0
MOVL C00039 V=800.0 PL=0
MOVL C00040 V=800.0 PL=0
MOVL C00041 V=800.0 PL=0
MOVL C00042 V=800.0 PL=0
MOVL C00043 V=800.0 PL=0
MOVL C00044 V=800.0 PL=0
MOVL C00045 V=800.0 PL=0
MOVL C00046 V=800.0 PL=0
MOVL C00047 V=800.0 PL=0
MOVL C00048 V=800.0 PL=0
MOVL C00049 V=800.0 PL=0
MOVL C00050 V=800.0 PL=0
MOVL C00051 V=800.0 PL=0
MOVL C00052 V=800.0 PL=0
MOVL C00053 V=800.0 PL=0
MOVL C00054 V=800.0 PL=0
MOVL C00055 V=800.0 PL=0
MOVL C00056 V=800.0 PL=0
MOVL C00057 V=800.0 PL=0
MOVL C00058 V=800.0 PL=0
MOVL C00059 V=800.0 PL=0
MOVL C00060 V=800.0 PL=0
MOVL C00061 V=800.0 PL=0
MOVL C00062 V=800.0 PL=0
MOVL C00063 V=800.0 PL=0
MOVL C00064 V=800.0 PL=0
MOVL C00065 V=800.0 PL=0
MOVL C00066 V=800.0 PL=0
MOVL C00067 V=800.0 PL=0
MOVL C00068 V=800.0 PL=0
MOVL C00069 V=800.0 PL=0
MOVL C00070 V=800.0 PL=0
MOVL C00071 V=800.0 PL=0
MOVL C00072 V=800.0 PL=0
MOVL C00073 V=800.0 PL=0
MOVL C00074 V=800.0 PL=0
MOVL C00075 V=800.0 PL=0
MOVL C00076 V=800.0 PL=0
MOVL C00077 V=800.0 PL=0
MOVL C00078 V=800.0 PL=0
MOVL C00079 V=800.0 PL=0
MOVL C00080 V=800.0 PL=0
MOVL C00081 V=800.0 PL=0
MOVL C00082 V=800.0 PL=0
MOVL C00083 V=800.0 PL=0
MOVL C00084 V=800.0 PL=0
MOVL C00085 V=800.0 PL=0
MOVL C00086 V=800.0 PL=0
MOVL C00087 V=800.0 PL=0
MOVL C00088 V=800.0 PL=0
MOVL C00089 V=800.0 PL=0
MOVL C00090 V=800.0 PL=0
MOVL C00091 V=800.0 PL=0
MOVL C00092 V=800.0 PL=0
MOVL C00093 V=800.0 PL=0
MOVL C00094 V=800.0 PL=0
MOVL C00095 V=800.0 PL=0
MOVL C00096 V=800.0 PL=0
MOVL C00097 V=800.0 PL=0
MOVL C00098 V=800.0 PL=0
MOVL C00099 V=800.0 PL=0
MOVL C00100 V=800.0 PL=0
MOVL C00101 V=800.0 PL=0
MOVL C00102 V=800.0 PL=0
MOVL C00103 V=800.0 PL=0
MOVL C00104 V=800.0 PL=0
MOVL C00105 V=800.0 PL=0
MOVL C00106 V=800.0 PL=0
MOVL C00107 V=800.0 PL=0
MOVL C00108 V=800.0 PL=0
MOVL C00109 V=800.0 PL=0
MOVL C00110 V=800.0 PL=0
MOVL C00111 V=800.0 PL=0
MOVL C00112 V=800.0 PL=0
MOVL C00113 V=800.0 PL=0
MOVL C00114 V=800.0 PL=0
MOVL C00115 V=800.0 PL=0
MOVL C00116 V=800.0 PL=0
MOVL C00117 V=800.0 PL=0
MOVL C00118 V=800.0 PL=0
MOVL C00119 V=800.0 PL=0
MOVL C00120 V=800.0 PL=0
MOVL C00121 V=800.0 PL=0
MOVL C00122 V=800.0 PL=0
MOVL C00123 V=800.0 PL=0
MOVL C00124 V=800.0 PL=0
MOVL C00125 V=800.0 PL=0
MOVL C00126 V=800.0 PL=0
MOVL C00127 V=800.0 PL=0
MOVL C00128 V=800.0 PL=0
MOVL C00129 V=800.0 PL=0
MOVL C00130 V=800.0 PL=0
MOVL C00131 V=800.0 PL=0
MOVL C00132 V=800.0 PL=0
MOVL C00133 V=800.0 PL=0
MOVL C00134 V=800.0 PL=0
MOVL C00135 V=800.0 PL=0
MOVL C00136 V=800.0 PL=0
MOVL C00137 V=800.0 PL=0
MOVL C00138 V=800.0 PL=0
MOVL C00139 V=800.0 PL=0
MOVL C00140 V=800.0 PL=0
MOVL C00141 V=800.0 PL=0
MOVL C00142 V=800.0 PL=0
MOVL C00143 V=800.0 PL=0
MOVL C00144 V=800.0 PL=0
MOVL C00145 V=800.0 PL=0
MOVL C00146 V=800.0 PL=0
MOVL C00147 V=800.0 PL=0
MOVL C00148 V=800.0 PL=0
MOVL C00149 V=800.0 PL=0
MOVL C00150 V=800.0 PL=0
MOVL C00151 V=800.0 PL=0
MOVL C00152 V=800.0 PL=0
MOVL C00153 V=800.0 PL=0
MOVL C00154 V=800.0 PL=0
MOVL C00155 V=800.0 PL=0
MOVL C00156 V=800.0 PL=0
MOVL C00157 V=800.0 PL=0
MOVL C00158 V=800.0 PL=0
MOVL C00159 V=800.0 PL=0
MOVL C00160 V=800.0 PL=0
MOVL C00161 V=800.0 PL=0
MOVL C00162 V=800.0 PL=0
MOVL C00163 V=800.0 PL=0
MOVL C00164 V=800.0 PL=0
MOVL C00165 V=800.0 PL=0
MOVL C00166 V=800.0 PL=0
MOVL C00167 V=800.0 PL=0
MOVL C00168 V=800.0 PL=0
MOVL C00169 V=800.0 PL=0
MOVL C00170 V=800.0 PL=0
MOVL C00171 V=800.0 PL=0
MOVL C00172 V=800.0 PL=0
MOVL C00173 V=800.0 PL=0
MOVL C00174 V=800.0 PL=0
MOVL C00175 V=800.0 PL=0
MOVL C00176 V=800.0 PL=0
MOVL C00177 V=800.0 PL=0
MOVL C00178 V=800.0 PL=0
MOVL C00179 V=800.0 PL=0
MOVL C00180 V=800.0 PL=0
MOVL C00181 V=800.0 PL=0
MOVL C00182 V=800.0 PL=0
MOVL C00183 V=800.0 PL=0
MOVL C00184 V=800.0 PL=0
MOVL C00185 V=800.0 PL=0
MOVL C00186 V=800.0 PL=0
MOVL C00187 V=800.0 PL=0
MOVL C00188 V=800.0 PL=0
MOVL C00189 V=800.0 PL=0
MOVL C00190 V=800.0 PL=0
MOVL C00191 V=800.0 PL=0
MOVL C00192 V=800.0 PL=0
MOVL C00193 V=800.0 PL=0
MOVL C00194 V=800.0 PL=0
MOVL C00195 V=800.0 PL=0
MOVL C00196 V=800.0 PL=0
MOVL C00197 V=800.0 PL=0
MOVL C00198 V=800.0 PL=0
MOVL C00199 V=800.0 PL=0
MOVL C00200 V=800.0 PL=0
MOVL C00201 V=800.0 PL=0
MOVL C00202 V=800.0 PL=0
MOVL C00203 V=800.0 PL=0
MOVL C00204 V=800.0 PL=0
MOVL C00205 V=800.0 PL=0
MOVL C00206 V=800.0 PL=0
MOVL C00207 V=800.0 PL=0
MOVL C00208 V=800.0 PL=0
MOVL C00209 V=800.0 PL=0
MOVL C00210 V=800.0 PL=0
MOVL C00211 V=800.0 PL=0
MOVL C00212 V=800.0 PL=0
MOVL C00213 V=800.0 PL=0
MOVL C00214 V=800.0 PL=0
MOVL C00215 V=800.0 PL=0
MOVL C00216 V=800.0 PL=0
MOVL C00217 V=800.0 PL=0
MOVL C00218 V=800.0 PL=0
MOVL C00219 V=800.0 PL=0
MOVL C00220 V=800.0 PL=0
MOVL C00221 V=800.0 PL=0
MOVL C00222 V=800.0 PL=0
MOVL C00223 V=800.0 PL=0
MOVL C00224 V=800.0 PL=0
MOVL C00225 V=800.0 PL=0
MOVL C00226 V=800.0 PL=0
MOVL C00227 V=800.0 PL=0
MOVL C00228 V=800.0 PL=0
MOVL C00229 V=800.0 PL=0
MOVL C00230 V=800.0 PL=0
MOVL C00231 V=800.0 PL=0
MOVL C00232 V=800.0 PL=0
MOVL C00233 V=800.0 PL=0
MOVL C00234 V=800.0 PL=0
MOVL C00235 V=800.0 PL=0
MOVL C00236 V=800.0 PL=0
MOVL C00237 V=800.0 PL=0
MOVL C00238 V=800.0 PL=0
MOVL C00239 V=800.0 PL=0
MOVL C00240 V=800.0 PL=0
MOVL C00241 V=800.0 PL=0
MOVL C00242 V=800.0 PL=0
MOVL C00243 V=800.0 PL=0
MOVL C00244 V=800.0 PL=0
MOVL C00245 V=800.0 PL=0
MOVL C00246 V=800.0 PL=0
MOVL C00247 V=800.0 PL=0
MOVL C00248 V=800.0 PL=0
MOVL C00249 V=800.0 PL=0
MOVL C00250 V=800.0 PL=0
MOVL C00251 V=800.0 PL=0
MOVL C00252 V=800.0 PL=0
MOVL C00253 V=800.0 PL=0
MOVL C00254 V=800.0 PL=0
MOVL C00255 V=800.0 PL=0
MOVL C00256 V=800.0 PL=0
MOVL C00257 V=800.0 PL=0
MOVL C00258 V=800.0 PL=0
MOVL C00259 V=800.0 PL=0
MOVL C00260 V=800.0 PL=0
MOVL C00261 V=800.0 PL=0
MOVL C00262 V=800.0 PL=0
MOVL C00263 V=800.0 PL=0
MOVL C00264 V=800.0 PL=0
MOVL C00265 V=800.0 PL=0
MOVL C00266 V=800.0 PL=0
MOVL C00267 V=800.0 PL=0
MOVL C00268 V=800.0 PL=0
MOVL C00269 V=800.0 PL=0
MOVL C00270 V=800.0 PL=0
MOVL C00271 V=800.0 PL=0
MOVL C00272 V=800.0 PL=0
MOVL C00273 V=800.0 PL=0
MOVL C00274 V=800.0 PL=0
MOVL C00275 V=800.0 PL=0
MOVL C00276 V=800.0 PL=0
MOVL C00277 V=800.0 PL=0
MOVL C00278 V=800.0 PL=0
MOVL C00279 V=800.0 PL=0
MOVL C00280 V=800.0 PL=0
MOVL C00281 V=800.0 PL=0
MOVL C00282 V=800.0 PL=0
MOVL C00283 V=800.0 PL=0
MOVL C00284 V=800.0 PL=0
MOVL C00285 V=800.0 PL=0
MOVL C00286 V=800.0 PL=0
MOVL C00287 V=800.0 PL=0
MOVL C00288 V=800.0 PL=0
MOVL C00289 V=800.0 PL=0
MOVL C00290 V=800.0 PL=0
MOVL C00291 V=800.0 PL=0
MOVL C00292 V=800.0 PL=0
MOVL C00293 V=800.0 PL=0
MOVL C00294 V=800.0 PL=0
MOVL C00295 V=800.0 PL=0
MOVL C00296 V=800.0 PL=0
MOVL C00297 V=800.0 PL=0
MOVL C00298 V=800.0 PL=0
MOVL C00299 V=800.0 PL=0
MOVL C00300 V=800.0 PL=0
MOVL C00301 V=800.0 PL=0
MOVL C00302 V=800.0 PL=0
MOVL C00303 V=800.0 PL=0
MOVL C00304 V=800.0 PL=0
MOVL C00305 V=800.0 PL=0
MOVL C00306 V=800.0 PL=0
MOVL C00307 V=800.0 PL=0
MOVL C00308 V=800.0 PL=0
MOVL C00309 V=800.0 PL=0
MOVL C00310 V=800.0 PL=0
MOVL C00311 V=800.0 PL=0
MOVL C00312 V=800.0 PL=0
MOVL C00313 V=800.0 PL=0
MOVL C00314 V=800.0 PL=0
MOVL C00315 V=800.0 PL=0
MOVL C00316 V=800.0 PL=0
MOVL C00317 V=800.0 PL=0
MOVL C00318 V=800.0 PL=0
MOVL C00319 V=800.0 PL=0
MOVL C00320 V=800.0 PL=0
MOVL C00321 V=800.0 PL=0
MOVL C00322 V=800.0 PL=0
MOVL C00323 V=800.0 PL=0
MOVL C00324 V=800.0 PL=0
MOVL C00325 V=800.0 PL=0
MOVL C00326 V=800.0 PL=0
MOVL C00327 V=800.0 PL=0
MOVL C00328 V=800.0 PL=0
MOVL C00329 V=800.0 PL=0
MOVL C00330 V=800.0 PL=0
MOVL C00331 V=800.0 PL=0
MOVL C00332 V=800.0 PL=0
MOVL C00333 V=800.0 PL=0
MOVL C00334 V=800.0 PL=0
MOVL C00335 V=800.0 PL=0
MOVL C00336 V=800.0 PL=0
MOVL C00337 V=800.0 PL=0
MOVL C00338 V=800.0 PL=0
MOVL C00339 V=800.0 PL=0
MOVL C00340 V=800.0 PL=0
MOVL C00341 V=800.0 PL=0
MOVL C00342 V=800.0 PL=0
MOVL C00343 V=800.0 PL=0
MOVL C00344 V=800.0 PL=0
MOVL C00345 V=800.0 PL=0
MOVL C00346 V=800.0 PL=0
MOVL C00347 V=800.0 PL=0
MOVL C00348 V=800.0 PL=0
MOVL C00349 V=800.0 PL=0
MOVL C00350 V=800.0 PL=0
MOVL C00351 V=800.0 PL=0
MOVL C00352 V=800.0 PL=0
MOVL C00353 V=800.0 PL=0
MOVL C00354 V=800.0 PL=0
MOVL C00355 V=800.0 PL=0
MOVL C00356 V=800.0 PL=0
MOVL C00357 V=800.0 PL=0
MOVL C00358 V=800.0 PL=0
MOVL C00359 V=800.0 PL=0
MOVL C00360 V=800.0 PL=0
MOVL C00361 V=800.0 PL=0
MOVL C00362 V=800.0 PL=0
MOVL C00363 V=800.0 PL=0
MOVL C00364 V=800.0 PL=0
MOVL C00365 V=800.0 PL=0
MOVL C00366 V=800.0 PL=0
MOVL C00367 V=800.0 PL=0
MOVL C00368 V=800.0 PL=0
MOVL C00369 V=800.0 PL=0
MOVL C00370 V=800.0 PL=0
MOVL C00371 V=800.0 PL=0
MOVL C00372 V=800.0 PL=0
MOVL C00373 V=800.0 PL=0
MOVL C00374 V=800.0 PL=0
MOVL C00375 V=800.0 PL=0
MOVL C00376 V=800.0 PL=0
MOVL C00377 V=800.0 PL=0
MOVL C00378 V=800.0 PL=0
MOVL C00379 V=800.0 PL=0
MOVL C00380 V=800.0 PL=0
MOVL C00381 V=800.0 PL=0
MOVL C00382 V=800.0 PL=0
MOVL C00383 V=800.0 PL=0
MOVL C00384 V=800.0 PL=0
MOVL C00385 V=800.0 PL=0
MOVL C00386 V=800.0 PL=0
MOVL C00387 V=800.0 PL=0
MOVL C00388 V=800.0 PL=0
MOVL C00389 V=800.0 PL=0
MOVL C00390 V=800.0 PL=0
MOVL C00391 V=800.0 PL=0
MOVL C00392 V=800.0 PL=0
MOVL C00393 V=800.0 PL=0
MOVL C00394 V=800.0 PL=0
MOVL C00395 V=800.0 PL=0
MOVL C00396 V=800.0 PL=0
MOVL C00397 V=800.0 PL=0
MOVL C00398 V=800.0 PL=0
MOVL C00399 V=800.0 PL=0
MOVL C00400 V=800.0 PL=0
MOVL C00401 V=800.0 PL=0
MOVL C00402 V=800.0 PL=0
MOVL C00403 V=800.0 PL=0
MOVL C00404 V=800.0 PL=0
MOVL C00405 V=800.0 PL=0
MOVL C00406 V=800.0 PL=0
MOVL C00407 V=800.0 PL=0
MOVL C00408 V=800.0 PL=0
MOVL C00409 V=800.0 PL=0
MOVL C00410 V=800.0 PL=0
MOVL C00411 V=800.0 PL=0
MOVL C00412 V=800.0 PL=0
MOVL C00413 V=800.0 PL=0
MOVL C00414 V=800.0 PL=0
MOVL C00415 V=800.0 PL=0
MOVL C00416 V=800.0 PL=0
MOVL C00417 V=800.0 PL=0
MOVL C00418 V=800.0 PL=0
MOVL C00419 V=800.0 PL=0
MOVL C00420 V=800.0 PL=0
MOVL C00421 V=800.0 PL=0
MOVL C00422 V=800.0 PL=0
MOVL C00423 V=800.0 PL=0
MOVL C00424 V=800.0 PL=0
MOVL C00425 V=800.0 PL=0
MOVL C00426 V=800.0 PL=0
MOVL C00427 V=800.0 PL=0
MOVL C00428 V=800.0 PL=0
MOVL C00429 V=800.0 PL=0
MOVL C00430 V=800.0 PL=0
MOVL C00431 V=800.0 PL=0
MOVL C00432 V=800.0 PL=0
MOVL C00433 V=800.0 PL=0
MOVL C00434 V=800.0 PL=0
MOVL C00435 V=800.0 PL=0
MOVL C00436 V=800.0 PL=0
MOVL C00437 V=800.0 PL=0
MOVL C00438 V=800.0 PL=0
MOVL C00439 V=800.0 PL=0
MOVL C00440 V=800.0 PL=0
MOVL C00441 V=800.0 PL=0
MOVL C00442 V=800.0 PL=0
MOVL C00443 V=800.0 PL=0
MOVL C00444 V=800.0 PL=0
MOVL C00445 V=800.0 PL=0
MOVL C00446 V=800.0 PL=0
MOVL C00447 V=800.0 PL=0
MOVL C00448 V=800.0 PL=0
MOVL C00449 V=800.0 PL=0
MOVL C00450 V=800.0 PL=0
MOVL C00451 V=800.0 PL=0
MOVL C00452 V=800.0 PL=0
MOVL C00453 V=800.0 PL=0
MOVL C00454 V=800.0 PL=0
MOVL C00455 V=800.0 PL=0
MOVL C00456 V=800.0 PL=0
MOVL C00457 V=800.0 PL=0
MOVL C00458 V=800.0 PL=0
MOVL C00459 V=800.0 PL=0
MOVL C00460 V=800.0 PL=0
MOVL C00461 V=800.0 PL=0
MOVL C00462 V=800.0 PL=0
MOVL C00463 V=800.0 PL=0
MOVL C00464 V=800.0 PL=0
MOVL C00465 V=800.0 PL=0
MOVL C00466 V=800.0 PL=0
MOVL C00467 V=800.0 PL=0
MOVL C00468 V=800.0 PL=0
MOVL C00469 V=800.0 PL=0
MOVL C00470 V=800.0 PL=0
MOVL C00471 V=800.0 PL=0
MOVL C00472 V=800.0 PL=0
MOVL C00473 V=800.0 PL=0
MOVL C00474 V=800.0 PL=0
MOVL C00475 V=800.0 PL=0
MOVL C00476 V=800.0 PL=0
MOVL C00477 V=800.0 PL=0
MOVL C00478 V=800.0 PL=0
MOVL C00479 V=800.0 PL=0
MOVL C00480 V=800.0 PL=0
MOVL C00481 V=800.0 PL=0
MOVL C00482 V=800.0 PL=0
MOVL C00483 V=800.0 PL=0
MOVL C00484 V=800.0 PL=0
MOVL C00485 V=800.0 PL=0
MOVL C00486 V=800.0 PL=0
MOVL C00487 V=800.0 PL=0
MOVL C00488 V=800.0 PL=0
MOVL C00489 V=800.0 PL=0
MOVL C00490 V=800.0 PL=0
MOVL C00491 V=800.0 PL=0
MOVL C00492 V=800.0 PL=0
MOVL C00493 V=800.0 PL=0
MOVL C00494 V=800.0 PL=0
MOVL C00495 V=800.0 PL=0
MOVL C00496 V=800.0 PL=0
MOVL C00497 V=800.0 PL=0
MOVL C00498 V=800.0 PL=0
MOVL C00499 V=800.0 PL=0
MOVL C00500 V=800.0 PL=0
MOVL C00501 V=800.0 PL=0
MOVL C00502 V=800.0 PL=0
MOVL C00503 V=800.0 PL=0
MOVL C00504 V=800.0 PL=0
MOVL C00505 V=800.0 PL=0
MOVL C00506 V=800.0 PL=0
MOVL C00507 V=800.0 PL=0
MOVL C00508 V=800.0 PL=0
MOVL C00509 V=800.0 PL=0
MOVL C00510 V=800.0 PL=0
MOVL C00511 V=800.0 PL=0
MOVL C00512 V=800.0 PL=0
MOVL C00513 V=800.0 PL=0
MOVL C00514 V=800.0 PL=0
MOVL C00515 V=800.0 PL=0
MOVL C00516 V=800.0 PL=0
MOVL C00517 V=800.0 PL=0
MOVL C00518 V=800.0 PL=0
MOVL C00519 V=800.0 PL=0
MOVL C00520 V=800.0 PL=0
MOVL C00521 V=800.0 PL=0
MOVL C00522 V=800.0 PL=0
MOVL C00523 V=800.0 PL=0
MOVL C00524 V=800.0 PL=0
MOVL C00525 V=800.0 PL=0
MOVL C00526 V=800.0 PL=0
MOVL C00527 V=800.0 PL=0
MOVL C00528 V=800.0 PL=0
MOVL C00529 V=800.0 PL=0
MOVL C00530 V=800.0 PL=0
MOVL C00531 V=800.0 PL=0
MOVL C00532 V=800.0 PL=0
MOVL C00533 V=800.0 PL=0
MOVL C00534 V=800.0 PL=0
MOVL C00535 V=800.0 PL=0
MOVL C00536 V=800.0 PL=0
MOVL C00537 V=800.0 PL=0
MOVL C00538 V=800.0 PL=0
MOVL C00539 V=800.0 PL=0
MOVL C00540 V=800.0 PL=0
MOVL C00541 V=800.0 PL=0
MOVL C00542 V=800.0 PL=0
MOVL C00543 V=800.0 PL=0
MOVL C00544 V=800.0 PL=0
MOVL C00545 V=800.0 PL=0
MOVL C00546 V=800.0 PL=0
MOVL C00547 V=800.0 PL=0
MOVL C00548 V=800.0 PL=0
MOVL C00549 V=800.0 PL=0
MOVL C00550 V=800.0 PL=0
MOVL C00551 V=800.0 PL=0
MOVL C00552 V=800.0 PL=0
MOVL C00553 V=800.0 PL=0
MOVL C00554 V=800.0 PL=0
MOVL C00555 V=800.0 PL=0
MOVL C00556 V=800.0 PL=0
MOVL C00557 V=800.0 PL=0
MOVL C00558 V=800.0 PL=0
MOVL C00559 V=800.0 PL=0
MOVL C00560 V=800.0 PL=0
MOVL C00561 V=800.0 PL=0
MOVL C00562 V=800.0 PL=0
MOVL C00563 V=800.0 PL=0
MOVL C00564 V=800.0 PL=0
MOVL C00565 V=800.0 PL=0
MOVL C00566 V=800.0 PL=0
MOVL C00567 V=800.0 PL=0
MOVL C00568 V=800.0 PL=0
MOVL C00569 V=800.0 PL=0
MOVL C00570 V=800.0 PL=0
MOVL C00571 V=800.0 PL=0
MOVL C00572 V=800.0 PL=0
MOVL C00573 V=800.0 PL=0
MOVL C00574 V=800.0 PL=0
MOVL C00575 V=800.0 PL=0
MOVL C00576 V=800.0 PL=0
MOVL C00577 V=800.0 PL=0
MOVL C00578 V=800.0 PL=0
MOVL C00579 V=800.0 PL=0
MOVL C00580 V=800.0 PL=0
MOVL C00581 V=800.0 PL=0
MOVL C00582 V=800.0 PL=0
MOVL C00583 V=800.0 PL=0
MOVL C00584 V=800.0 PL=0
MOVL C00585 V=800.0 PL=0
MOVL C00586 V=800.0 PL=0
MOVL C00587 V=800.0 PL=0
MOVL C00588 V=800.0 PL=0
MOVL C00589 V=800.0 PL=0
MOVL C00590 V=800.0 PL=0
MOVL C00591 V=800.0 PL=0
MOVL C00592 V=800.0 PL=0
MOVL C00593 V=800.0 PL=0
MOVL C00594 V=800.0 PL=0
MOVL C00595 V=800.0 PL=0
MOVL C00596 V=800.0 PL=0
MOVL C00597 V=800.0 PL=0
MOVL C00598 V=800.0 PL=0
MOVL C00599 V=800.0 PL=0
MOVL C00600 V=800.0 PL=0
MOVL C00601 V=800.0 PL=0
MOVL C00602 V=800.0 PL=0
MOVL C00603 V=800.0 PL=0
MOVL C00604 V=800.0 PL=0
MOVL C00605 V=800.0 PL=0
MOVL C00606 V=800.0 PL=0
MOVL C00607 V=800.0 PL=0
MOVL C00608 V=800.0 PL=0
MOVL C00609 V=800.0 PL=0
MOVL C00610 V=800.0 PL=0
MOVL C00611 V=800.0 PL=0
MOVL C00612 V=800.0 PL=0
MOVL C00613 V=800.0 PL=0
MOVL C00614 V=800.0 PL=0
MOVL C00615 V=800.0 PL=0
MOVL C00616 V=800.0 PL=0
MOVL C00617 V=800.0 PL=0
MOVL C00618 V=800.0 PL=0
MOVL C00619 V=800.0 PL=0
MOVL C00620 V=800.0 PL=0
MOVL C00621 V=800.0 PL=0
MOVL C00622 V=800.0 PL=0
MOVL C00623 V=800.0 PL=0
MOVL C00624 V=800.0 PL=0
MOVL C00625 V=800.0 PL=0
MOVL C00626 V=800.0 PL=0
MOVL C00627 V=800.0 PL=0
MOVL C00628 V=800.0 PL=0
MOVL C00629 V=800.0 PL=0
MOVL C00630 V=800.0 PL=0
MOVL C00631 V=800.0 PL=0
MOVL C00632 V=800.0 PL=0
MOVL C00633 V=800.0 PL=0
MOVL C00634 V=800.0 PL=0
MOVL C00635 V=800.0 PL=0
MOVL C00636 V=800.0 PL=0
MOVL C00637 V=800.0 PL=0
MOVL C00638 V=800.0 PL=0
MOVL C00639 V=800.0 PL=0
MOVL C00640 V=800.0 PL=0
MOVL C00641 V=800.0 PL=0
MOVL C00642 V=800.0 PL=0
MOVL C00643 V=800.0 PL=0
MOVL C00644 V=800.0 PL=0
MOVL C00645 V=800.0 PL=0
MOVL C00646 V=800.0 PL=0
MOVL C00647 V=800.0 PL=0
MOVL C00648 V=800.0 PL=0
MOVL C00649 V=800.0 PL=0
MOVL C00650 V=800.0 PL=0
MOVL C00651 V=800.0 PL=0
MOVL C00652 V=800.0 PL=0
MOVL C00653 V=800.0 PL=0
MOVL C00654 V=800.0 PL=0
MOVL C00655 V=800.0 PL=0
MOVL C00656 V=800.0 PL=0
MOVL C00657 V=800.0 PL=0
MOVL C00658 V=800.0 PL=0
MOVL C00659 V=800.0 PL=0
MOVL C00660 V=800.0 PL=0
MOVL C00661 V=800.0 PL=0
MOVL C00662 V=800.0 PL=0
MOVL C00663 V=800.0 PL=0
MOVL C00664 V=800.0 PL=0
MOVL C00665 V=800.0 PL=0
MOVL C00666 V=800.0 PL=0
MOVL C00667 V=800.0 PL=0
MOVL C00668 V=800.0 PL=0
MOVL C00669 V=800.0 PL=0
MOVL C00670 V=800.0 PL=0
MOVL C00671 V=800.0 PL=0
MOVL C00672 V=800.0 PL=0
MOVL C00673 V=800.0 PL=0
MOVL C00674 V=800.0 PL=0
MOVL C00675 V=800.0 PL=0
MOVL C00676 V=800.0 PL=0
MOVL C00677 V=800.0 PL=0
MOVL C00678 V=800.0 PL=0
MOVL C00679 V=800.0 PL=0
MOVL C00680 V=800.0 PL=0
MOVL C00681 V=800.0 PL=0
MOVL C00682 V=800.0 PL=0
MOVL C00683 V=800.0 PL=0
MOVL C00684 V=800.0 PL=0
MOVL C00685 V=800.0 PL=0
MOVL C00686 V=800.0 PL=0
MOVL C00687 V=800.0 PL=0
MOVL C00688 V=800.0 PL=0
MOVL C00689 V=800.0 PL=0
MOVL C00690 V=800.0 PL=0
MOVL C00691 V=800.0 PL=0
MOVL C00692 V=800.0 PL=0
MOVL C00693 V=800.0 PL=0
MOVL C00694 V=800.0 PL=0
MOVL C00695 V=800.0 PL=0
MOVL C00696 V=800.0 PL=0
MOVL C00697 V=800.0 PL=0
MOVL C00698 V=800.0 PL=0
MOVL C00699 V=800.0 PL=0
MOVL C00700 V=800.0 PL=0
MOVL C00701 V=800.0 PL=0
MOVL C00702 V=800.0 PL=0
MOVL C00703 V=800.0 PL=0
MOVL C00704 V=800.0 PL=0
MOVL C00705 V=800.0 PL=0
MOVL C00706 V=800.0 PL=0
MOVL C00707 V=800.0 PL=0
MOVL C00708 V=800.0 PL=0
MOVL C00709 V=800.0 PL=0
MOVL C00710 V=800.0 PL=0
MOVL C00711 V=800.0 PL=0
MOVL C00712 V=800.0 PL=0
MOVL C00713 V=800.0 PL=0
MOVL C00714 V=800.0 PL=0
MOVL C00715 V=800.0 PL=0
MOVL C00716 V=800.0 PL=0
MOVL C00717 V=800.0 PL=0
MOVL C00718 V=800.0 PL=0
MOVL C00719 V=800.0 PL=0
MOVL C00720 V=800.0 PL=0
MOVL C00721 V=800.0 PL=0
MOVL C00722 V=800.0 PL=0
MOVL C00723 V=800.0 PL=0
MOVL C00724 V=800.0 PL=0
MOVL C00725 V=800.0 PL=0
MOVL C00726 V=800.0 PL=0
MOVL C00727 V=800.0 PL=0
MOVL C00728 V=800.0 PL=0
MOVL C00729 V=800.0 PL=0
MOVL C00730 V=800.0 PL=0
MOVL C00731 V=800.0 PL=0
MOVL C00732 V=800.0 PL=0
MOVL C00733 V=800.0 PL=0
MOVL C00734 V=800.0 PL=0
MOVL C00735 V=800.0 PL=0
MOVL C00736 V=800.0 PL=0
MOVL C00737 V=800.0 PL=0
MOVL C00738 V=800.0 PL=0
MOVL C00739 V=800.0 PL=0
MOVL C00740 V=800.0 PL=0
MOVL C00741 V=800.0 PL=0
MOVL C00742 V=800.0 PL=0
MOVL C00743 V=800.0 PL=0
MOVL C00744 V=800.0 PL=0
MOVL C00745 V=800.0 PL=0
MOVL C00746 V=800.0 PL=0
MOVL C00747 V=800.0 PL=0
MOVL C00748 V=800.0 PL=0
MOVL C00749 V=800.0 PL=0
MOVL C00750 V=800.0 PL=0
MOVL C00751 V=800.0 PL=0
MOVL C00752 V=800.0 PL=0
MOVL C00753 V=800.0 PL=0
MOVL C00754 V=800.0 PL=0
MOVL C00755 V=800.0 PL=0
MOVL C00756 V=800.0 PL=0
MOVL C00757 V=800.0 PL=0
MOVL C00758 V=800.0 PL=0
MOVL C00759 V=800.0 PL=0
MOVL C00760 V=800.0 PL=0
MOVL C00761 V=800.0 PL=0
MOVL C00762 V=800.0 PL=0
MOVL C00763 V=800.0 PL=0
MOVL C00764 V=800.0 PL=0
MOVL C00765 V=800.0 PL=0
MOVL C00766 V=800.0 PL=0
MOVL C00767 V=800.0 PL=0
MOVL C00768 V=800.0 PL=0
MOVL C00769 V=800.0 PL=0
MOVL C00770 V=800.0 PL=0
MOVL C00771 V=800.0 PL=0
MOVL C00772 V=800.0 PL=0
MOVL C00773 V=800.0 PL=0
MOVL C00774 V=800.0 PL=0
MOVL C00775 V=800.0 PL=0
MOVL C00776 V=800.0 PL=0
MOVL C00777 V=800.0 PL=0
MOVL C00778 V=800.0 PL=0
MOVL C00779 V=800.0 PL=0
MOVL C00780 V=800.0 PL=0
MOVL C00781 V=800.0 PL=0
MOVL C00782 V=800.0 PL=0
MOVL C00783 V=800.0 PL=0
MOVL C00784 V=800.0 PL=0
MOVL C00785 V=800.0 PL=0
MOVL C00786 V=800.0 PL=0
MOVL C00787 V=800.0 PL=0
MOVL C00788 V=800.0 PL=0
MOVL C00789 V=800.0 PL=0
MOVL C00790 V=800.0 PL=0
MOVL C00791 V=800.0 PL=0
MOVL C00792 V=800.0 PL=0
MOVL C00793 V=800.0 PL=0
MOVL C00794 V=800.0 PL=0
MOVL C00795 V=800.0 PL=0
MOVL C00796 V=800.0 PL=0
MOVL C00797 V=800.0 PL=0
MOVL C00798 V=800.0 PL=0
MOVL C00799 V=800.0 PL=0
MOVL C00800 V=800.0 PL=0
MOVL C00801 V=800.0 PL=0
MOVL C00802 V=800.0 PL=0
MOVL C00803 V=800.0 PL=0
MOVL C00804 V=800.0 PL=0
MOVL C00805 V=800.0 PL=0
MOVL C00806 V=800.0 PL=0
MOVL C00807 V=800.0 PL=0
MOVL C00808 V=800.0 PL=0
MOVL C00809 V=800.0 PL=0
MOVL C00810 V=800.0 PL=0
MOVL C00811 V=800.0 PL=0
MOVL C00812 V=800.0 PL=0
MOVL C00813 V=800.0 PL=0
MOVL C00814 V=800.0 PL=0
MOVL C00815 V=800.0 PL=0
MOVL C00816 V=800.0 PL=0
MOVL C00817 V=800.0 PL=0
MOVL C00818 V=800.0 PL=0
MOVL C00819 V=800.0 PL=0
MOVL C00820 V=800.0 PL=0
MOVL C00821 V=800.0 PL=0
MOVL C00822 V=800.0 PL=0
MOVL C00823 V=800.0 PL=0
MOVL C00824 V=800.0 PL=0
MOVL C00825 V=800.0 PL=0
MOVL C00826 V=800.0 PL=0
MOVL C00827 V=800.0 PL=0
MOVL C00828 V=800.0 PL=0
MOVL C00829 V=800.0 PL=0
MOVL C00830 V=800.0 PL=0
MOVL C00831 V=800.0 PL=0
MOVL C00832 V=800.0 PL=0
MOVL C00833 V=800.0 PL=0
MOVL C00834 V=800.0 PL=0
MOVL C00835 V=800.0 PL=0
MOVL C00836 V=800.0 PL=0
MOVL C00837 V=800.0 PL=0
MOVL C00838 V=800.0 PL=0
MOVL C00839 V=800.0 PL=0
MOVL C00840 V=800.0 PL=0
MOVL C00841 V=800.0 PL=0
MOVL C00842 V=800.0 PL=0
MOVL C00843 V=800.0 PL=0
MOVL C00844 V=800.0 PL=0
MOVL C00845 V=800.0 PL=0
MOVL C00846 V=800.0 PL=0
MOVL C00847 V=800.0 PL=0
MOVL C00848 V=800.0 PL=0
MOVL C00849 V=800.0 PL=0
MOVL C00850 V=800.0 PL=0
MOVL C00851 V=800.0 PL=0
MOVL C00852 V=800.0 PL=0
MOVL C00853 V=800.0 PL=0
MOVL C00854 V=800.0 PL=0
MOVL C00855 V=800.0 PL=0
MOVL C00856 V=800.0 PL=0
MOVL C00857 V=800.0 PL=0
MOVL C00858 V=800.0 PL=0
MOVL C00859 V=800.0 PL=0
MOVL C00860 V=800.0 PL=0
MOVL C00861 V=800.0 PL=0
MOVL C00862 V=800.0 PL=0
MOVL C00863 V=800.0 PL=0
MOVL C00864 V=800.0 PL=0
MOVL C00865 V=800.0 PL=0
MOVL C00866 V=800.0 PL=0
MOVL C00867 V=800.0 PL=0
MOVL C00868 V=800.0 PL=0
MOVL C00869 V=800.0 PL=0
MOVL C00870 V=800.0 PL=0
MOVL C00871 V=800.0 PL=0
MOVL C00872 V=800.0 PL=0
MOVL C00873 V=800.0 PL=0
MOVL C00874 V=800.0 PL=0
MOVL C00875 V=800.0 PL=0
MOVL C00876 V=800.0 PL=0
MOVL C00877 V=800.0 PL=0
MOVL C00878 V=800.0 PL=0
MOVL C00879 V=800.0 PL=0
MOVL C00880 V=800.0 PL=0
MOVL C00881 V=800.0 PL=0
MOVL C00882 V=800.0 PL=0
MOVL C00883 V=800.0 PL=0
MOVL C00884 V=800.0 PL=0
MOVL C00885 V=800.0 PL=0
MOVL C00886 V=800.0 PL=0
MOVL C00887 V=800.0 PL=0
MOVL C00888 V=800.0 PL=0
MOVL C00889 V=800.0 PL=0
MOVL C00890 V=800.0 PL=0
MOVL C00891 V=800.0 PL=0
MOVL C00892 V=800.0 PL=0
MOVL C00893 V=800.0 PL=0
MOVL C00894 V=800.0 PL=0
MOVL C00895 V=800.0 PL=0
MOVL C00896 V=800.0 PL=0
MOVL C00897 V=800.0 PL=0
MOVL C00898 V=800.0 PL=0
MOVL C00899 V=800.0 PL=0
MOVL C00900 V=800.0 PL=0
MOVL C00901 V=800.0 PL=0
MOVL C00902 V=800.0 PL=0
MOVL C00903 V=800.0 PL=0
MOVL C00904 V=800.0 PL=0
MOVL C00905 V=800.0 PL=0
MOVL C00906 V=800.0 PL=0
MOVL C00907 V=800.0 PL=0
MOVL C00908 V=800.0 PL=0
MOVL C00909 V=800.0 PL=0
MOVL C00910 V=800.0 PL=0
MOVL C00911 V=800.0 PL=0
MOVL C00912 V=800.0 PL=0
MOVL C00913 V=800.0 PL=0
MOVL C00914 V=800.0 PL=0
MOVL C00915 V=800.0 PL=0
MOVL C00916 V=800.0 PL=0
MOVL C00917 V=800.0 PL=0
MOVL C00918 V=800.0 PL=0
MOVL C00919 V=800.0 PL=0
MOVL C00920 V=800.0 PL=0
MOVL C00921 V=800.0 PL=0
MOVL C00922 V=800.0 PL=0
MOVL C00923 V=800.0 PL=0
MOVL C00924 V=800.0 PL=0
MOVL C00925 V=800.0 PL=0
MOVL C00926 V=800.0 PL=0
MOVL C00927 V=800.0 PL=0
MOVL C00928 V=800.0 PL=0
MOVL C00929 V=800.0 PL=0
MOVL C00930 V=800.0 PL=0
MOVL C00931 V=800.0 PL=0
MOVL C00932 V=800.0 PL=0
MOVL C00933 V=800.0 PL=0
MOVL C00934 V=800.0 PL=0
MOVL C00935 V=800.0 PL=0
MOVL C00936 V=800.0 PL=0
MOVL C00937 V=800.0 PL=0
MOVL C00938 V=800.0 PL=0
MOVL C00939 V=800.0 PL=0
MOVL C00940 V=800.0 PL=0
MOVL C00941 V=800.0 PL=0
MOVL C00942 V=800.0 PL=0
MOVL C00943 V=800.0 PL=0
MOVL C00944 V=800.0 PL=0
MOVL C00945 V=800.0 PL=0
MOVL C00946 V=800.0 PL=0
MOVL C00947 V=800.0 PL=0
MOVL C00948 V=800.0 PL=0
MOVL C00949 V=800.0 PL=0
MOVL C00950 V=800.0 PL=0
MOVL C00951 V=800.0 PL=0
MOVL C00952 V=800.0 PL=0
MOVL C00953 V=800.0 PL=0
MOVL C00954 V=800.0 PL=0
MOVL C00955 V=800.0 PL=0
MOVL C00956 V=800.0 PL=0
MOVL C00957 V=800.0 PL=0
MOVL C00958 V=800.0 PL=0
MOVL C00959 V=800.0 PL=0
MOVL C00960 V=800.0 PL=0
MOVL C00961 V=800.0 PL=0
MOVL C00962 V=800.0 PL=0
MOVL C00963 V=800.0 PL=0
MOVL C00964 V=800.0 PL=0
MOVL C00965 V=800.0 PL=0
MOVL C00966 V=800.0 PL=0
MOVL C00967 V=800.0 PL=0
MOVL C00968 V=800.0 PL=0
MOVL C00969 V=800.0 PL=0
MOVL C00970 V=800.0 PL=0
MOVL C00971 V=800.0 PL=0
MOVL C00972 V=800.0 PL=0
MOVL C00973 V=800.0 PL=0
MOVL C00974 V=800.0 PL=0
MOVL C00975 V=800.0 PL=0
MOVL C00976 V=800.0 PL=0
MOVL C00977 V=800.0 PL=0
MOVL C00978 V=800.0 PL=0
MOVL C00979 V=800.0 PL=0
MOVL C00980 V=800.0 PL=0
MOVL C00981 V=800.0 PL=0
MOVL C00982 V=800.0 PL=0
MOVL C00983 V=800.0 PL=0
MOVL C00984 V=800.0 PL=0
MOVL C00985 V=800.0 PL=0
MOVL C00986 V=800.0 PL=0
MOVL C00987 V=800.0 PL=0
MOVL C00988 V=800.0 PL=0
MOVL C00989 V=800.0 PL=0
MOVL C00990 V=800.0 PL=0
MOVL C00991 V=800.0 PL=0
MOVL C00992 V=800.0 PL=0
MOVL C00993 V=800.0 PL=0
MOVL C00994 V=800.0 PL=0
MOVL C00995 V=800.0 PL=0
MOVL C00996 V=800.0 PL=0
MOVL C00997 V=800.0 PL=0
MOVL C00998 V=800.0 PL=0
MOVL C00999 V=800.0 PL=0
MOVL C01000 V=800.0 PL=0
MOVL C01001 V=800.0 PL=0
MOVL C01002 V=800.0 PL=0
MOVL C01003 V=800.0 PL=0
MOVL C01004 V=800.0 PL=0
MOVL C01005 V=800.0 PL=0
MOVL C01006 V=800.0 PL=0
MOVL C01007 V=800.0 PL=0
MOVL C01008 V=800.0 PL=0
MOVL C01009 V=800.0 PL=0
MOVL C01010 V=800.0 PL=0
MOVL C01011 V=800.0 PL=0
MOVL C01012 V=800.0 PL=0
MOVL C01013 V=800.0 PL=0
MOVL C01014 V=800.0 PL=0
MOVL C01015 V=800.0 PL=0
MOVL C01016 V=800.0 PL=0
MOVL C01017 V=800.0 PL=0
MOVL C01018 V=800.0 PL=0
MOVL C01019 V=800.0 PL=0
MOVL C01020 V=800.0 PL=0
MOVL C01021 V=800.0 PL=0
MOVL C01022 V=800.0 PL=0
MOVL C01023 V=800.0 PL=0
MOVL C01024 V=800.0 PL=0
MOVL C01025 V=800.0 PL=0
MOVL C01026 V=800.0 PL=0
MOVL C01027 V=800.0 PL=0
MOVL C01028 V=800.0 PL=0
MOVL C01029 V=800.0 PL=0
MOVL C01030 V=800.0 PL=0
MOVL C01031 V=800.0 PL=0
MOVL C01032 V=800.0 PL=0
MOVL C01033 V=800.0 PL=0
MOVL C01034 V=800.0 PL=0
MOVL C01035 V=800.0 PL=0
MOVL C01036 V=800.0 PL=0
MOVL C01037 V=800.0 PL=0
MOVL C01038 V=800.0 PL=0
MOVL C01039 V=800.0 PL=0
MOVL C01040 V=800.0 PL=0
MOVL C01041 V=800.0 PL=0
MOVL C01042 V=800.0 PL=0
MOVL C01043 V=800.0 PL=0
MOVL C01044 V=800.0 PL=0
MOVL C01045 V=800.0 PL=0
MOVL C01046 V=800.0 PL=0
MOVL C01047 V=800.0 PL=0
MOVL C01048 V=800.0 PL=0
MOVL C01049 V=800.0 PL=0
MOVL C01050 V=800.0 PL=0
MOVL C01051 V=800.0 PL=0
MOVL C01052 V=800.0 PL=0
MOVL C01053 V=800.0 PL=0
MOVL C01054 V=800.0 PL=0
MOVL C01055 V=800.0 PL=0
MOVL C01056 V=800.0 PL=0
MOVL C01057 V=800.0 PL=0
MOVL C01058 V=800.0 PL=0
MOVL C01059 V=800.0 PL=0
MOVL C01060 V=800.0 PL=0
MOVL C01061 V=800.0 PL=0
MOVL C01062 V=800.0 PL=0
MOVL C01063 V=800.0 PL=0
MOVL C01064 V=800.0 PL=0
MOVL C01065 V=800.0 PL=0
MOVL C01066 V=800.0 PL=0
MOVL C01067 V=800.0 PL=0
MOVL C01068 V=800.0 PL=0
MOVL C01069 V=800.0 PL=0
MOVL C01070 V=800.0 PL=0
MOVL C01071 V=800.0 PL=0
MOVL C01072 V=800.0 PL=0
MOVL C01073 V=800.0 PL=0
MOVL C01074 V=800.0 PL=0
MOVL C01075 V=800.0 PL=0
MOVL C01076 V=800.0 PL=0
MOVL C01077 V=800.0 PL=0
MOVL C01078 V=800.0 PL=0
MOVL C01079 V=800.0 PL=0
MOVL C01080 V=800.0 PL=0
MOVL C01081 V=800.0 PL=0
MOVL C01082 V=800.0 PL=0
MOVL C01083 V=800.0 PL=0
MOVL C01084 V=800.0 PL=0
MOVL C01085 V=800.0 PL=0
MOVL C01086 V=800.0 PL=0
MOVL C01087 V=800.0 PL=0
MOVL C01088 V=800.0 PL=0
MOVL C01089 V=800.0 PL=0
MOVL C01090 V=800.0 PL=0
MOVL C01091 V=800.0 PL=0
MOVL C01092 V=800.0 PL=0
MOVL C01093 V=800.0 PL=0
MOVL C01094 V=800.0 PL=0
MOVL C01095 V=800.0 PL=0
MOVL C01096 V=800.0 PL=0
MOVL C01097 V=800.0 PL=0
MOVL C01098 V=800.0 PL=0
MOVL C01099 V=800.0 PL=0
MOVL C01100 V=800.0 PL=0
MOVL C01101 V=800.0 PL=0
MOVL C01102 V=800.0 PL=0
MOVL C01103 V=800.0 PL=0
MOVL C01104 V=800.0 PL=0
MOVL C01105 V=800.0 PL=0
MOVL C01106 V=800.0 PL=0
MOVL C01107 V=800.0 PL=0
MOVL C01108 V=800.0 PL=0
MOVL C01109 V=800.0 PL=0
MOVL C01110 V=800.0 PL=0
MOVL C01111 V=800.0 PL=0
MOVL C01112 V=800.0 PL=0
MOVL C01113 V=800.0 PL=0
MOVL C01114 V=800.0 PL=0
MOVL C01115 V=800.0 PL=0
MOVL C01116 V=800.0 PL=0
MOVL C01117 V=800.0 PL=0
MOVL C01118 V=800.0 PL=0
MOVL C01119 V=800.0 PL=0
MOVL C01120 V=800.0 PL=0
MOVL C01121 V=800.0 PL=0
MOVL C01122 V=800.0 PL=0
MOVL C01123 V=800.0 PL=0
MOVL C01124 V=800.0 PL=0
MOVL C01125 V=800.0 PL=0
MOVL C01126 V=800.0 PL=0
MOVL C01127 V=800.0 PL=0
MOVL C01128 V=800.0 PL=0
MOVL C01129 V=800.0 PL=0
MOVL C01130 V=800.0 PL=0
MOVL C01131 V=800.0 PL=0
MOVL C01132 V=800.0 PL=0
MOVL C01133 V=800.0 PL=0
MOVL C01134 V=800.0 PL=0
MOVL C01135 V=800.0 PL=0
MOVL C01136 V=800.0 PL=0
MOVL C01137 V=800.0 PL=0
MOVL C01138 V=800.0 PL=0
MOVL C01139 V=800.0 PL=0
MOVL C01140 V=800.0 PL=0
MOVL C01141 V=800.0 PL=0
MOVL C01142 V=800.0 PL=0
MOVL C01143 V=800.0 PL=0
MOVL C01144 V=800.0 PL=0
MOVL C01145 V=800.0 PL=0
MOVL C01146 V=800.0 PL=0
MOVL C01147 V=800.0 PL=0
MOVL C01148 V=800.0 PL=0
MOVL C01149 V=800.0 PL=0
MOVL C01150 V=800.0 PL=0
MOVL C01151 V=800.0 PL=0
MOVL C01152 V=800.0 PL=0
MOVL C01153 V=800.0 PL=0
MOVL C01154 V=800.0 PL=0
MOVL C01155 V=800.0 PL=0
MOVL C01156 V=800.0 PL=0
MOVL C01157 V=800.0 PL=0
MOVL C01158 V=800.0 PL=0
MOVL C01159 V=800.0 PL=0
MOVL C01160 V=800.0 PL=0
MOVL C01161 V=800.0 PL=0
MOVL C01162 V=800.0 PL=0
MOVL C01163 V=800.0 PL=0
MOVL C01164 V=800.0 PL=0
MOVL C01165 V=800.0 PL=0
MOVL C01166 V=800.0 PL=0
MOVL C01167 V=800.0 PL=0
MOVL C01168 V=800.0 PL=0
MOVL C01169 V=800.0 PL=0
MOVL C01170 V=800.0 PL=0
MOVL C01171 V=800.0 PL=0
MOVL C01172 V=800.0 PL=0
MOVL C01173 V=800.0 PL=0
MOVL C01174 V=800.0 PL=0
MOVL C01175 V=800.0 PL=0
MOVL C01176 V=800.0 PL=0
MOVL C01177 V=800.0 PL=0
MOVL C01178 V=800.0 PL=0
MOVL C01179 V=800.0 PL=0
MOVL C01180 V=800.0 PL=0
MOVL C01181 V=800.0 PL=0
MOVL C01182 V=800.0 PL=0
MOVL C01183 V=800.0 PL=0
MOVL C01184 V=800.0 PL=0
MOVL C01185 V=800.0 PL=0
MOVL C01186 V=800.0 PL=0
MOVL C01187 V=800.0 PL=0
MOVL C01188 V=800.0 PL=0
MOVL C01189 V=800.0 PL=0
MOVL C01190 V=800.0 PL=0
MOVL C01191 V=800.0 PL=0
MOVL C01192 V=800.0 PL=0
MOVL C01193 V=800.0 PL=0
MOVL C01194 V=800.0 PL=0
MOVL C01195 V=800.0 PL=0
MOVL C01196 V=800.0 PL=0
MOVL C01197 V=800.0 PL=0
MOVL C01198 V=800.0 PL=0
MOVL C01199 V=800.0 PL=0
MOVL C01200 V=800.0 PL=0
MOVL C01201 V=800.0 PL=0
MOVL C01202 V=800.0 PL=0
MOVL C01203 V=800.0 PL=0
MOVL C01204 V=800.0 PL=0
MOVL C01205 V=800.0 PL=0
MOVL C01206 V=800.0 PL=0
MOVL C01207 V=800.0 PL=0
MOVL C01208 V=800.0 PL=0
MOVL C01209 V=800.0 PL=0
MOVL C01210 V=800.0 PL=0
MOVL C01211 V=800.0 PL=0
MOVL C01212 V=800.0 PL=0
MOVL C01213 V=800.0 PL=0
MOVL C01214 V=800.0 PL=0
MOVL C01215 V=800.0 PL=0
MOVL C01216 V=800.0 PL=0
MOVL C01217 V=800.0 PL=0
MOVL C01218 V=800.0 PL=0
MOVL C01219 V=800.0 PL=0
MOVL C01220 V=800.0 PL=0
MOVL C01221 V=800.0 PL=0
MOVL C01222 V=800.0 PL=0
MOVL C01223 V=800.0 PL=0
MOVL C01224 V=800.0 PL=0
MOVL C01225 V=800.0 PL=0
MOVL C01226 V=800.0 PL=0
MOVL C01227 V=800.0 PL=0
MOVL C01228 V=800.0 PL=0
MOVL C01229 V=800.0 PL=0
MOVL C01230 V=800.0 PL=0
MOVL C01231 V=800.0 PL=0
MOVL C01232 V=800.0 PL=0
MOVL C01233 V=800.0 PL=0
MOVL C01234 V=800.0 PL=0
MOVL C01235 V=800.0 PL=0
MOVL C01236 V=800.0 PL=0
MOVL C01237 V=800.0 PL=0
MOVL C01238 V=800.0 PL=0
MOVL C01239 V=800.0 PL=0
MOVL C01240 V=800.0 PL=0
MOVL C01241 V=800.0 PL=0
MOVL C01242 V=800.0 PL=0
MOVL C01243 V=800.0 PL=0
MOVL C01244 V=800.0 PL=0
MOVL C01245 V=800.0 PL=0
MOVL C01246 V=800.0 PL=0
MOVL C01247 V=800.0 PL=0
MOVL C01248 V=800.0 PL=0
MOVL C01249 V=800.0 PL=0
MOVL C01250 V=800.0 PL=0
MOVL C01251 V=800.0 PL=0
MOVL C01252 V=800.0 PL=0
MOVL C01253 V=800.0 PL=0
MOVL C01254 V=800.0 PL=0
MOVL C01255 V=800.0 PL=0
MOVL C01256 V=800.0 PL=0
MOVL C01257 V=800.0 PL=0
MOVL C01258 V=800.0 PL=0
MOVL C01259 V=800.0 PL=0
MOVL C01260 V=800.0 PL=0
MOVL C01261 V=800.0 PL=0
MOVL C01262 V=800.0 PL=0
MOVL C01263 V=800.0 PL=0
MOVL C01264 V=800.0 PL=0
MOVL C01265 V=800.0 PL=0
MOVL C01266 V=800.0 PL=0
MOVL C01267 V=800.0 PL=0
MOVL C01268 V=800.0 PL=0
MOVL C01269 V=800.0 PL=0
MOVL C01270 V=800.0 PL=0
MOVL C01271 V=800.0 PL=0
MOVL C01272 V=800.0 PL=0
MOVL C01273 V=800.0 PL=0
MOVL C01274 V=800.0 PL=0
MOVL C01275 V=800.0 PL=0
MOVL C01276 V=800.0 PL=0
MOVL C01277 V=800.0 PL=0
MOVL C01278 V=800.0 PL=0
MOVL C01279 V=800.0 PL=0
MOVL C01280 V=800.0 PL=0
MOVL C01281 V=800.0 PL=0
MOVL C01282 V=800.0 PL=0
MOVL C01283 V=800.0 PL=0
MOVL C01284 V=800.0 PL=0
MOVL C01285 V=800.0 PL=0
MOVL C01286 V=800.0 PL=0
MOVL C01287 V=800.0 PL=0
MOVL C01288 V=800.0 PL=0
MOVL C01289 V=800.0 PL=0
MOVL C01290 V=800.0 PL=0
MOVL C01291 V=800.0 PL=0
MOVL C01292 V=800.0 PL=0
MOVL C01293 V=800.0 PL=0
MOVL C01294 V=800.0 PL=0
MOVL C01295 V=800.0 PL=0
MOVL C01296 V=800.0 PL=0
MOVL C01297 V=800.0 PL=0
MOVL C01298 V=800.0 PL=0
MOVL C01299 V=800.0 PL=0
MOVL C01300 V=800.0 PL=0
MOVL C01301 V=800.0 PL=0
MOVL C01302 V=800.0 PL=0
MOVL C01303 V=800.0 PL=0
MOVL C01304 V=800.0 PL=0
MOVL C01305 V=800.0 PL=0
MOVL C01306 V=800.0 PL=0
MOVL C01307 V=800.0 PL=0
MOVL C01308 V=800.0 PL=0
MOVL C01309 V=800.0 PL=0
MOVL C01310 V=800.0 PL=0
MOVL C01311 V=800.0 PL=0
MOVL C01312 V=800.0 PL=0
MOVL C01313 V=800.0 PL=0
MOVL C01314 V=800.0 PL=0
MOVL C01315 V=800.0 PL=0
MOVL C01316 V=800.0 PL=0
MOVL C01317 V=800.0 PL=0
MOVL C01318 V=800.0 PL=0
MOVL C01319 V=800.0 PL=0
MOVL C01320 V=800.0 PL=0
MOVL C01321 V=800.0 PL=0
MOVL C01322 V=800.0 PL=0
MOVL C01323 V=800.0 PL=0
MOVL C01324 V=800.0 PL=0
MOVL C01325 V=800.0 PL=0
MOVL C01326 V=800.0 PL=0
MOVL C01327 V=800.0 PL=0
MOVL C01328 V=800.0 PL=0
MOVL C01329 V=800.0 PL=0
MOVL C01330 V=800.0 PL=0
MOVL C01331 V=800.0 PL=0
MOVL C01332 V=800.0 PL=0
MOVL C01333 V=800.0 PL=0
MOVL C01334 V=800.0 PL=0
MOVL C01335 V=800.0 PL=0
MOVL C01336 V=800.0 PL=0
MOVL C01337 V=800.0 PL=0
MOVL C01338 V=800.0 PL=0
MOVL C01339 V=800.0 PL=0
MOVL C01340 V=800.0 PL=0
MOVL C01341 V=800.0 PL=0
MOVL C01342 V=800.0 PL=0
MOVL C01343 V=800.0 PL=0
MOVL C01344 V=800.0 PL=0
MOVL C01345 V=800.0 PL=0
MOVL C01346 V=800.0 PL=0
MOVL C01347 V=800.0 PL=0
MOVL C01348 V=800.0 PL=0
MOVL C01349 V=800.0 PL=0
MOVL C01350 V=800.0 PL=0
MOVL C01351 V=800.0 PL=0
MOVL C01352 V=800.0 PL=0
MOVL C01353 V=800.0 PL=0
MOVL C01354 V=800.0 PL=0
MOVL C01355 V=800.0 PL=0
MOVL C01356 V=800.0 PL=0
MOVL C01357 V=800.0 PL=0
MOVL C01358 V=800.0 PL=0
MOVL C01359 V=800.0 PL=0
MOVL C01360 V=800.0 PL=0
MOVL C01361 V=800.0 PL=0
MOVL C01362 V=800.0 PL=0
MOVL C01363 V=800.0 PL=0
MOVL C01364 V=800.0 PL=0
MOVL C01365 V=800.0 PL=0
MOVL C01366 V=800.0 PL=0
MOVL C01367 V=800.0 PL=0
MOVL C01368 V=800.0 PL=0
MOVL C01369 V=800.0 PL=0
MOVL C01370 V=800.0 PL=0
MOVL C01371 V=800.0 PL=0
MOVL C01372 V=800.0 PL=0
MOVL C01373 V=800.0 PL=0
MOVL C01374 V=800.0 PL=0
MOVL C01375 V=800.0 PL=0
MOVL C01376 V=800.0 PL=0
MOVL C01377 V=800.0 PL=0
MOVL C01378 V=800.0 PL=0
MOVL C01379 V=800.0 PL=0
MOVL C01380 V=800.0 PL=0
MOVL C01381 V=800.0 PL=0
MOVL C01382 V=800.0 PL=0
MOVL C01383 V=800.0 PL=0
MOVL C01384 V=800.0 PL=0
MOVL C01385 V=800.0 PL=0
MOVL C01386 V=800.0 PL=0
MOVL C01387 V=800.0 PL=0
MOVL C01388 V=800.0 PL=0
MOVL C01389 V=800.0 PL=0
MOVL C01390 V=800.0 PL=0
MOVL C01391 V=800.0 PL=0
MOVL C01392 V=800.0 PL=0
MOVL C01393 V=800.0 PL=0
MOVL C01394 V=800.0 PL=0
MOVL C01395 V=800.0 PL=0
MOVL C01396 V=800.0 PL=0
MOVL C01397 V=800.0 PL=0
MOVL C01398 V=800.0 PL=0
MOVL C01399 V=800.0 PL=0
MOVL C01400 V=800.0 PL=0
MOVL C01401 V=800.0 PL=0
MOVL C01402 V=800.0 PL=0
MOVL C01403 V=800.0 PL=0
MOVL C01404 V=800.0 PL=0
MOVL C01405 V=800.0 PL=0
MOVL C01406 V=800.0 PL=0
MOVL C01407 V=800.0 PL=0
MOVL C01408 V=800.0 PL=0
MOVL C01409 V=800.0 PL=0
MOVL C01410 V=800.0 PL=0
MOVL C01411 V=800.0 PL=0
MOVL C01412 V=800.0 PL=0
MOVL C01413 V=800.0 PL=0
MOVL C01414 V=800.0 PL=0
MOVL C01415 V=800.0 PL=0
MOVL C01416 V=800.0 PL=0
MOVL C01417 V=800.0 PL=0
MOVL C01418 V=800.0 PL=0
MOVL C01419 V=800.0 PL=0
MOVL C01420 V=800.0 PL=0
MOVL C01421 V=800.0 PL=0
MOVL C01422 V=800.0 PL=0
MOVL C01423 V=800.0 PL=0
MOVL C01424 V=800.0 PL=0
MOVL C01425 V=800.0 PL=0
MOVL C01426 V=800.0 PL=0
MOVL C01427 V=800.0 PL=0
MOVL C01428 V=800.0 PL=0
MOVL C01429 V=800.0 PL=0
MOVL C01430 V=800.0 PL=0
MOVL C01431 V=800.0 PL=0
MOVL C01432 V=800.0 PL=0
MOVL C01433 V=800.0 PL=0
MOVL C01434 V=800.0 PL=0
MOVL C01435 V=800.0 PL=0
MOVL C01436 V=800.0 PL=0
MOVL C01437 V=800.0 PL=0
MOVL C01438 V=800.0 PL=0
MOVL C01439 V=800.0 PL=0
MOVL C01440 V=800.0 PL=0
MOVL C01441 V=800.0 PL=0
MOVL C01442 V=800.0 PL=0
MOVL C01443 V=800.0 PL=0
MOVL C01444 V=800.0 PL=0
MOVL C01445 V=800.0 PL=0
MOVL C01446 V=800.0 PL=0
MOVL C01447 V=800.0 PL=0
MOVL C01448 V=800.0 PL=0
MOVL C01449 V=800.0 PL=0
MOVL C01450 V=800.0 PL=0
MOVL C01451 V=800.0 PL=0
MOVL C01452 V=800.0 PL=0
MOVL C01453 V=800.0 PL=0
MOVL C01454 V=800.0 PL=0
MOVL C01455 V=800.0 PL=0
MOVL C01456 V=800.0 PL=0
MOVL C01457 V=800.0 PL=0
MOVL C01458 V=800.0 PL=0
MOVL C01459 V=800.0 PL=0
MOVL C01460 V=800.0 PL=0
MOVL C01461 V=800.0 PL=0
MOVL C01462 V=800.0 PL=0
MOVL C01463 V=800.0 PL=0
MOVL C01464 V=800.0 PL=0
MOVL C01465 V=800.0 PL=0
MOVL C01466 V=800.0 PL=0
MOVL C01467 V=800.0 PL=0
MOVL C01468 V=800.0 PL=0
MOVL C01469 V=800.0 PL=0
MOVL C01470 V=800.0 PL=0
MOVL C01471 V=800.0 PL=0
MOVL C01472 V=800.0 PL=0
MOVL C01473 V=800.0 PL=0
MOVL C01474 V=800.0 PL=0
MOVL C01475 V=800.0 PL=0
MOVL C01476 V=800.0 PL=0
MOVL C01477 V=800.0 PL=0
MOVL C01478 V=800.0 PL=0
MOVL C01479 V=800.0 PL=0
MOVL C01480 V=800.0 PL=0
MOVL C01481 V=800.0 PL=0
MOVL C01482 V=800.0 PL=0
MOVL C01483 V=800.0 PL=0
MOVL C01484 V=800.0 PL=0
MOVL C01485 V=800.0 PL=0
MOVL C01486 V=800.0 PL=0
MOVL C01487 V=800.0 PL=0
MOVL C01488 V=800.0 PL=0
MOVL C01489 V=800.0 PL=0
MOVL C01490 V=800.0 PL=0
MOVL C01491 V=800.0 PL=0
MOVL C01492 V=800.0 PL=0
MOVL C01493 V=800.0 PL=0
MOVL C01494 V=800.0 PL=0
MOVL C01495 V=800.0 PL=0
MOVL C01496 V=800.0 PL=0
MOVL C01497 V=800.0 PL=0
MOVL C01498 V=800.0 PL=0
MOVL C01499 V=800.0 PL=0
MOVL C01500 V=800.0 PL=0
MOVL C01501 V=800.0 PL=0
MOVL C01502 V=800.0 PL=0
MOVL C01503 V=800.0 PL=0
MOVL C01504 V=800.0 PL=0
MOVL C01505 V=800.0 PL=0
MOVL C01506 V=800.0 PL=0
MOVL C01507 V=800.0 PL=0
MOVL C01508 V=800.0 PL=0
MOVL C01509 V=800.0 PL=0
MOVL C01510 V=800.0 PL=0
MOVL C01511 V=800.0 PL=0
MOVL C01512 V=800.0 PL=0
MOVL C01513 V=800.0 PL=0
MOVL C01514 V=800.0 PL=0
MOVL C01515 V=800.0 PL=0
MOVL C01516 V=800.0 PL=0
MOVL C01517 V=800.0 PL=0
MOVL C01518 V=800.0 PL=0
MOVL C01519 V=800.0 PL=0
MOVL C01520 V=800.0 PL=0
MOVL C01521 V=800.0 PL=0
MOVL C01522 V=800.0 PL=0
MOVL C01523 V=800.0 PL=0
MOVL C01524 V=800.0 PL=0
MOVL C01525 V=800.0 PL=0
MOVL C01526 V=800.0 PL=0
MOVL C01527 V=800.0 PL=0
MOVL C01528 V=800.0 PL=0
MOVL C01529 V=800.0 PL=0
MOVL C01530 V=800.0 PL=0
MOVL C01531 V=800.0 PL=0
MOVL C01532 V=800.0 PL=0
MOVL C01533 V=800.0 PL=0
MOVL C01534 V=800.0 PL=0
MOVL C01535 V=800.0 PL=0
MOVL C01536 V=800.0 PL=0
MOVL C01537 V=800.0 PL=0
MOVL C01538 V=800.0 PL=0
MOVL C01539 V=800.0 PL=0
MOVL C01540 V=800.0 PL=0
MOVL C01541 V=800.0 PL=0
MOVL C01542 V=800.0 PL=0
MOVL C01543 V=800.0 PL=0
MOVL C01544 V=800.0 PL=0
MOVL C01545 V=800.0 PL=0
MOVL C01546 V=800.0 PL=0
MOVL C01547 V=800.0 PL=0
MOVL C01548 V=800.0 PL=0
MOVL C01549 V=800.0 PL=0
MOVL C01550 V=800.0 PL=0
MOVL C01551 V=800.0 PL=0
MOVL C01552 V=800.0 PL=0
MOVL C01553 V=800.0 PL=0
MOVL C01554 V=800.0 PL=0
MOVL C01555 V=800.0 PL=0
MOVL C01556 V=800.0 PL=0
MOVL C01557 V=800.0 PL=0
MOVL C01558 V=800.0 PL=0
MOVL C01559 V=800.0 PL=0
MOVL C01560 V=800.0 PL=0
MOVL C01561 V=800.0 PL=0
MOVL C01562 V=800.0 PL=0
MOVL C01563 V=800.0 PL=0
MOVL C01564 V=800.0 PL=0
MOVL C01565 V=800.0 PL=0
MOVL C01566 V=800.0 PL=0
MOVL C01567 V=800.0 PL=0
MOVL C01568 V=800.0 PL=0
MOVL C01569 V=800.0 PL=0
MOVL C01570 V=800.0 PL=0
MOVL C01571 V=800.0 PL=0
MOVL C01572 V=800.0 PL=0
MOVL C01573 V=800.0 PL=0
MOVL C01574 V=800.0 PL=0
MOVL C01575 V=800.0 PL=0
MOVL C01576 V=800.0 PL=0
MOVL C01577 V=800.0 PL=0
MOVL C01578 V=800.0 PL=0
MOVL C01579 V=800.0 PL=0
MOVL C01580 V=800.0 PL=0
MOVL C01581 V=800.0 PL=0
MOVL C01582 V=800.0 PL=0
MOVL C01583 V=800.0 PL=0
MOVL C01584 V=800.0 PL=0
MOVL C01585 V=800.0 PL=0
MOVL C01586 V=800.0 PL=0
MOVL C01587 V=800.0 PL=0
MOVL C01588 V=800.0 PL=0
MOVL C01589 V=800.0 PL=0
MOVL C01590 V=800.0 PL=0
MOVL C01591 V=800.0 PL=0
MOVL C01592 V=800.0 PL=0
MOVL C01593 V=800.0 PL=0
MOVL C01594 V=800.0 PL=0
MOVL C01595 V=800.0 PL=0
MOVL C01596 V=800.0 PL=0
MOVL C01597 V=800.0 PL=0
MOVL C01598 V=800.0 PL=0
MOVL C01599 V=800.0 PL=0
MOVL C01600 V=800.0 PL=0
MOVL C01601 V=800.0 PL=0
MOVL C01602 V=800.0 PL=0
MOVL C01603 V=800.0 PL=0
MOVL C01604 V=800.0 PL=0
MOVL C01605 V=800.0 PL=0
MOVL C01606 V=800.0 PL=0
MOVL C01607 V=800.0 PL=0
MOVL C01608 V=800.0 PL=0
MOVL C01609 V=800.0 PL=0
MOVL C01610 V=800.0 PL=0
MOVL C01611 V=800.0 PL=0
MOVL C01612 V=800.0 PL=0
MOVL C01613 V=800.0 PL=0
MOVL C01614 V=800.0 PL=0
MOVL C01615 V=800.0 PL=0
MOVL C01616 V=800.0 PL=0
MOVL C01617 V=800.0 PL=0
MOVL C01618 V=800.0 PL=0
MOVL C01619 V=800.0 PL=0
MOVL C01620 V=800.0 PL=0
MOVL C01621 V=800.0 PL=0
MOVL C01622 V=800.0 PL=0
MOVL C01623 V=800.0 PL=0
MOVL C01624 V=800.0 PL=0
MOVL C01625 V=800.0 PL=0
MOVL C01626 V=800.0 PL=0
MOVL C01627 V=800.0 PL=0
MOVL C01628 V=800.0 PL=0
MOVL C01629 V=800.0 PL=0
MOVL C01630 V=800.0 PL=0
MOVL C01631 V=800.0 PL=0
MOVL C01632 V=800.0 PL=0
MOVL C01633 V=800.0 PL=0
MOVL C01634 V=800.0 PL=0
MOVL C01635 V=800.0 PL=0
MOVL C01636 V=800.0 PL=0
MOVL C01637 V=800.0 PL=0
MOVL C01638 V=800.0 PL=0
MOVL C01639 V=800.0 PL=0
MOVL C01640 V=800.0 PL=0
MOVL C01641 V=800.0 PL=0
MOVL C01642 V=800.0 PL=0
MOVL C01643 V=800.0 PL=0
MOVL C01644 V=800.0 PL=0
MOVL C01645 V=800.0 PL=0
MOVL C01646 V=800.0 PL=0
MOVL C01647 V=800.0 PL=0
MOVL C01648 V=800.0 PL=0
MOVL C01649 V=800.0 PL=0
MOVL C01650 V=800.0 PL=0
MOVL C01651 V=800.0 PL=0
MOVL C01652 V=800.0 PL=0
MOVL C01653 V=800.0 PL=0
MOVL C01654 V=800.0 PL=0
MOVL C01655 V=800.0 PL=0
MOVL C01656 V=800.0 PL=0
MOVL C01657 V=800.0 PL=0
MOVL C01658 V=800.0 PL=0
MOVL C01659 V=800.0 PL=0
MOVL C01660 V=800.0 PL=0
MOVL C01661 V=800.0 PL=0
MOVL C01662 V=800.0 PL=0
MOVL C01663 V=800.0 PL=0
MOVL C01664 V=800.0 PL=0
MOVL C01665 V=800.0 PL=0
MOVL C01666 V=800.0 PL=0
MOVL C01667 V=800.0 PL=0
MOVL C01668 V=800.0 PL=0
MOVL C01669 V=800.0 PL=0
MOVL C01670 V=800.0 PL=0
MOVL C01671 V=800.0 PL=0
MOVL C01672 V=800.0 PL=0
MOVL C01673 V=800.0 PL=0
MOVL C01674 V=800.0 PL=0
MOVL C01675 V=800.0 PL=0
MOVL C01676 V=800.0 PL=0
MOVL C01677 V=800.0 PL=0
MOVL C01678 V=800.0 PL=0
MOVL C01679 V=800.0 PL=0
MOVL C01680 V=800.0 PL=0
MOVL C01681 V=800.0 PL=0
MOVL C01682 V=800.0 PL=0
MOVL C01683 V=800.0 PL=0
MOVL C01684 V=800.0 PL=0
MOVL C01685 V=800.0 PL=0
MOVL C01686 V=800.0 PL=0
MOVL C01687 V=800.0 PL=0
MOVL C01688 V=800.0 PL=0
MOVL C01689 V=800.0 PL=0
MOVL C01690 V=800.0 PL=0
MOVL C01691 V=800.0 PL=0
MOVL C01692 V=800.0 PL=0
MOVL C01693 V=800.0 PL=0
MOVL C01694 V=800.0 PL=0
MOVL C01695 V=800.0 PL=0
MOVL C01696 V=800.0 PL=0
MOVL C01697 V=800.0 PL=0
MOVL C01698 V=800.0 PL=0
MOVL C01699 V=800.0 PL=0
MOVL C01700 V=800.0 PL=0
MOVL C01701 V=800.0 PL=0
MOVL C01702 V=800.0 PL=0
MOVL C01703 V=800.0 PL=0
MOVL C01704 V=800.0 PL=0
MOVL C01705 V=800.0 PL=0
MOVL C01706 V=800.0 PL=0
MOVL C01707 V=800.0 PL=0
MOVL C01708 V=800.0 PL=0
MOVL C01709 V=800.0 PL=0
MOVL C01710 V=800.0 PL=0
MOVL C01711 V=800.0 PL=0
MOVL C01712 V=800.0 PL=0
MOVL C01713 V=800.0 PL=0
MOVL C01714 V=800.0 PL=0
MOVL C01715 V=800.0 PL=0
MOVL C01716 V=800.0 PL=0
MOVL C01717 V=800.0 PL=0
MOVL C01718 V=800.0 PL=0
MOVL C01719 V=800.0 PL=0
MOVL C01720 V=800.0 PL=0
MOVL C01721 V=800.0 PL=0
MOVL C01722 V=800.0 PL=0
MOVL C01723 V=800.0 PL=0
MOVL C01724 V=800.0 PL=0
MOVL C01725 V=800.0 PL=0
MOVL C01726 V=800.0 PL=0
MOVL C01727 V=800.0 PL=0
MOVL C01728 V=800.0 PL=0
MOVL C01729 V=800.0 PL=0
MOVL C01730 V=800.0 PL=0
MOVL C01731 V=800.0 PL=0
MOVL C01732 V=800.0 PL=0
MOVL C01733 V=800.0 PL=0
MOVL C01734 V=800.0 PL=0
MOVL C01735 V=800.0 PL=0
MOVL C01736 V=800.0 PL=0
MOVL C01737 V=800.0 PL=0
MOVL C01738 V=800.0 PL=0
MOVL C01739 V=800.0 PL=0
MOVL C01740 V=800.0 PL=0
MOVL C01741 V=800.0 PL=0
MOVL C01742 V=800.0 PL=0
MOVL C01743 V=800.0 PL=0
MOVL C01744 V=800.0 PL=0
MOVL C01745 V=800.0 PL=0
MOVL C01746 V=800.0 PL=0
MOVL C01747 V=800.0 PL=0
MOVL C01748 V=800.0 PL=0
MOVL C01749 V=800.0 PL=0
MOVL C01750 V=800.0 PL=0
MOVL C01751 V=800.0 PL=0
MOVL C01752 V=800.0 PL=0
MOVL C01753 V=800.0 PL=0
MOVL C01754 V=800.0 PL=0
MOVL C01755 V=800.0 PL=0
MOVL C01756 V=800.0 PL=0
MOVL C01757 V=800.0 PL=0
MOVL C01758 V=800.0 PL=0
MOVL C01759 V=800.0 PL=0
MOVL C01760 V=800.0 PL=0
MOVL C01761 V=800.0 PL=0
MOVL C01762 V=800.0 PL=0
MOVL C01763 V=800.0 PL=0
MOVL C01764 V=800.0 PL=0
MOVL C01765 V=800.0 PL=0
MOVL C01766 V=800.0 PL=0
MOVL C01767 V=800.0 PL=0
MOVL C01768 V=800.0 PL=0
MOVL C01769 V=800.0 PL=0
MOVL C01770 V=800.0 PL=0
MOVL C01771 V=800.0 PL=0
MOVL C01772 V=800.0 PL=0
MOVL C01773 V=800.0 PL=0
MOVL C01774 V=800.0 PL=0
MOVL C01775 V=800.0 PL=0
MOVL C01776 V=800.0 PL=0
MOVL C01777 V=800.0 PL=0
MOVL C01778 V=800.0 PL=0
MOVL C01779 V=800.0 PL=0
MOVL C01780 V=800.0 PL=0
MOVL C01781 V=800.0 PL=0
MOVL C01782 V=800.0 PL=0
MOVL C01783 V=800.0 PL=0
MOVL C01784 V=800.0 PL=0
MOVL C01785 V=800.0 PL=0
MOVL C01786 V=800.0 PL=0
MOVL C01787 V=800.0 PL=0
MOVL C01788 V=800.0 PL=0
MOVL C01789 V=800.0 PL=0
MOVL C01790 V=800.0 PL=0
MOVL C01791 V=800.0 PL=0
MOVL C01792 V=800.0 PL=0
MOVL C01793 V=800.0 PL=0
MOVL C01794 V=800.0 PL=0
MOVL C01795 V=800.0 PL=0
MOVL C01796 V=800.0 PL=0
MOVL C01797 V=800.0 PL=0
MOVL C01798 V=800.0 PL=0
MOVL C01799 V=800.0 PL=0
MOVL C01800 V=800.0 PL=0
MOVL C01801 V=800.0 PL=0
MOVL C01802 V=800.0 PL=0
MOVL C01803 V=800.0 PL=0
MOVL C01804 V=800.0 PL=0
MOVL C01805 V=800.0 PL=0
MOVL C01806 V=800.0 PL=0
MOVL C01807 V=800.0 PL=0
MOVL C01808 V=800.0 PL=0
MOVL C01809 V=800.0 PL=0
MOVL C01810 V=800.0 PL=0
MOVL C01811 V=800.0 PL=0
MOVL C01812 V=800.0 PL=0
MOVL C01813 V=800.0 PL=0
MOVL C01814 V=800.0 PL=0
MOVL C01815 V=800.0 PL=0
MOVL C01816 V=800.0 PL=0
MOVL C01817 V=800.0 PL=0
MOVL C01818 V=800.0 PL=0
MOVL C01819 V=800.0 PL=0
MOVL C01820 V=800.0 PL=0
MOVL C01821 V=800.0 PL=0
MOVL C01822 V=800.0 PL=0
MOVL C01823 V=800.0 PL=0
MOVL C01824 V=800.0 PL=0
MOVL C01825 V=800.0 PL=0
MOVL C01826 V=800.0 PL=0
MOVL C01827 V=800.0 PL=0
MOVL C01828 V=800.0 PL=0
MOVL C01829 V=800.0 PL=0
MOVL C01830 V=800.0 PL=0
MOVL C01831 V=800.0 PL=0
MOVL C01832 V=800.0 PL=0
MOVL C01833 V=800.0 PL=0
MOVL C01834 V=800.0 PL=0
MOVL C01835 V=800.0 PL=0
MOVL C01836 V=800.0 PL=0
MOVL C01837 V=800.0 PL=0
MOVL C01838 V=800.0 PL=0
MOVL C01839 V=800.0 PL=0
MOVL C01840 V=800.0 PL=0
MOVL C01841 V=800.0 PL=0
MOVL C01842 V=800.0 PL=0
MOVL C01843 V=800.0 PL=0
MOVL C01844 V=800.0 PL=0
MOVL C01845 V=800.0 PL=0
MOVL C01846 V=800.0 PL=0
MOVL C01847 V=800.0 PL=0
MOVL C01848 V=800.0 PL=0
MOVL C01849 V=800.0 PL=0
MOVL C01850 V=800.0 PL=0
MOVL C01851 V=800.0 PL=0
MOVL C01852 V=800.0 PL=0
MOVL C01853 V=800.0 PL=0
MOVL C01854 V=800.0 PL=0
MOVL C01855 V=800.0 PL=0
MOVL C01856 V=800.0 PL=0
MOVL C01857 V=800.0 PL=0
MOVL C01858 V=800.0 PL=0
MOVL C01859 V=800.0 PL=0
MOVL C01860 V=800.0 PL=0
MOVL C01861 V=800.0 PL=0
MOVL C01862 V=800.0 PL=0
MOVL C01863 V=800.0 PL=0
MOVL C01864 V=800.0 PL=0
MOVL C01865 V=800.0 PL=0
MOVL C01866 V=800.0 PL=0
MOVL C01867 V=800.0 PL=0
MOVL C01868 V=800.0 PL=0
MOVL C01869 V=800.0 PL=0
MOVL C01870 V=800.0 PL=0
MOVL C01871 V=800.0 PL=0
MOVL C01872 V=800.0 PL=0
MOVL C01873 V=800.0 PL=0
MOVL C01874 V=800.0 PL=0
MOVL C01875 V=800.0 PL=0
MOVL C01876 V=800.0 PL=0
MOVL C01877 V=800.0 PL=0
MOVL C01878 V=800.0 PL=0
MOVL C01879 V=800.0 PL=0
MOVL C01880 V=800.0 PL=0
MOVL C01881 V=800.0 PL=0
MOVL C01882 V=800.0 PL=0
MOVL C01883 V=800.0 PL=0
MOVL C01884 V=800.0 PL=0
MOVL C01885 V=800.0 PL=0
MOVL C01886 V=800.0 PL=0
MOVL C01887 V=800.0 PL=0
MOVL C01888 V=800.0 PL=0
MOVL C01889 V=800.0 PL=0
MOVL C01890 V=800.0 PL=0
MOVL C01891 V=800.0 PL=0
MOVL C01892 V=800.0 PL=0
MOVL C01893 V=800.0 PL=0
MOVL C01894 V=800.0 PL=0
MOVL C01895 V=800.0 PL=0
MOVL C01896 V=800.0 PL=0
MOVL C01897 V=800.0 PL=0
MOVL C01898 V=800.0 PL=0
MOVL C01899 V=800.0 PL=0
MOVL C01900 V=800.0 PL=0
MOVL C01901 V=800.0 PL=0
MOVL C01902 V=800.0 PL=0
MOVL C01903 V=800.0 PL=0
MOVL C01904 V=800.0 PL=0
MOVL C01905 V=800.0 PL=0
MOVL C01906 V=800.0 PL=0
MOVL C01907 V=800.0 PL=0
MOVL C01908 V=800.0 PL=0
MOVL C01909 V=800.0 PL=0
MOVL C01910 V=800.0 PL=0
MOVL C01911 V=800.0 PL=0
MOVL C01912 V=800.0 PL=0
MOVL C01913 V=800.0 PL=0
MOVL C01914 V=800.0 PL=0
MOVL C01915 V=800.0 PL=0
MOVL C01916 V=800.0 PL=0
MOVL C01917 V=800.0 PL=0
MOVL C01918 V=800.0 PL=0
MOVL C01919 V=800.0 PL=0
MOVL C01920 V=800.0 PL=0
MOVL C01921 V=800.0 PL=0
MOVL C01922 V=800.0 PL=0
MOVL C01923 V=800.0 PL=0
MOVL C01924 V=800.0 PL=0
MOVL C01925 V=800.0 PL=0
MOVL C01926 V=800.0 PL=0
MOVL C01927 V=800.0 PL=0
MOVL C01928 V=800.0 PL=0
MOVL C01929 V=800.0 PL=0
MOVL C01930 V=800.0 PL=0
MOVL C01931 V=800.0 PL=0
MOVL C01932 V=800.0 PL=0
MOVL C01933 V=800.0 PL=0
MOVL C01934 V=800.0 PL=0
MOVL C01935 V=800.0 PL=0
MOVL C01936 V=800.0 PL=0
MOVL C01937 V=800.0 PL=0
MOVL C01938 V=800.0 PL=0
MOVL C01939 V=800.0 PL=0
MOVL C01940 V=800.0 PL=0
MOVL C01941 V=800.0 PL=0
MOVL C01942 V=800.0 PL=0
MOVL C01943 V=800.0 PL=0
MOVL C01944 V=800.0 PL=0
MOVL C01945 V=800.0 PL=0
MOVL C01946 V=800.0 PL=0
MOVL C01947 V=800.0 PL=0
MOVL C01948 V=800.0 PL=0
MOVL C01949 V=800.0 PL=0
MOVL C01950 V=800.0 PL=0
MOVL C01951 V=800.0 PL=0
MOVL C01952 V=800.0 PL=0
MOVL C01953 V=800.0 PL=0
MOVL C01954 V=800.0 PL=0
MOVL C01955 V=800.0 PL=0
MOVL C01956 V=800.0 PL=0
MOVL C01957 V=800.0 PL=0
MOVL C01958 V=800.0 PL=0
MOVL C01959 V=800.0 PL=0
MOVL C01960 V=800.0 PL=0
MOVL C01961 V=800.0 PL=0
MOVL C01962 V=800.0 PL=0
MOVL C01963 V=800.0 PL=0
MOVL C01964 V=800.0 PL=0
MOVL C01965 V=800.0 PL=0
MOVL C01966 V=800.0 PL=0
MOVL C01967 V=800.0 PL=0
MOVL C01968 V=800.0 PL=0
MOVL C01969 V=800.0 PL=0
MOVL C01970 V=800.0 PL=0
MOVL C01971 V=800.0 PL=0
MOVL C01972 V=800.0 PL=0
MOVL C01973 V=800.0 PL=0
MOVL C01974 V=800.0 PL=0
MOVL C01975 V=800.0 PL=0
MOVL C01976 V=800.0 PL=0
MOVL C01977 V=800.0 PL=0
MOVL C01978 V=800.0 PL=0
MOVL C01979 V=800.0 PL=0
MOVL C01980 V=800.0 PL=0
MOVL C01981 V=800.0 PL=0
MOVL C01982 V=800.0 PL=0
MOVL C01983 V=800.0 PL=0
MOVL C01984 V=800.0 PL=0
MOVL C01985 V=800.0 PL=0
MOVL C01986 V=800.0 PL=0
MOVL C01987 V=800.0 PL=0
MOVL C01988 V=800.0 PL=0
MOVL C01989 V=800.0 PL=0
MOVL C01990 V=800.0 PL=0
MOVL C01991 V=800.0 PL=0
MOVL C01992 V=800.0 PL=0
MOVL C01993 V=800.0 PL=0
MOVL C01994 V=800.0 PL=0
MOVL C01995 V=800.0 PL=0
MOVL C01996 V=800.0 PL=0
MOVL C01997 V=800.0 PL=0
MOVL C01998 V=800.0 PL=0
MOVL C01999 V=800.0 PL=0
MOVL C02000 V=800.0 PL=0
MOVL C02001 V=800.0 PL=0
MOVL C02002 V=800.0 PL=0
MOVL C02003 V=800.0 PL=0
MOVL C02004 V=800.0 PL=0
MOVL C02005 V=800.0 PL=0
MOVL C02006 V=800.0 PL=0
MOVL C02007 V=800.0 PL=0
MOVL C02008 V=800.0 PL=0
MOVL C02009 V=800.0 PL=0
MOVL C02010 V=800.0 PL=0
MOVL C02011 V=800.0 PL=0
MOVL C02012 V=800.0 PL=0
MOVL C02013 V=800.0 PL=0
MOVL C02014 V=800.0 PL=0
MOVL C02015 V=800.0 PL=0
MOVL C02016 V=800.0 PL=0
MOVL C02017 V=800.0 PL=0
MOVL C02018 V=800.0 PL=0
MOVL C02019 V=800.0 PL=0
MOVL C02020 V=800.0 PL=0
MOVL C02021 V=800.0 PL=0
MOVL C02022 V=800.0 PL=0
MOVL C02023 V=800.0 PL=0
MOVL C02024 V=800.0 PL=0
MOVL C02025 V=800.0 PL=0
MOVL C02026 V=800.0 PL=0
MOVL C02027 V=800.0 PL=0
MOVL C02028 V=800.0 PL=0
MOVL C02029 V=800.0 PL=0
MOVL C02030 V=800.0 PL=0
MOVL C02031 V=800.0 PL=0
MOVL C02032 V=800.0 PL=0
MOVL C02033 V=800.0 PL=0
MOVL C02034 V=800.0 PL=0
MOVL C02035 V=800.0 PL=0
MOVL C02036 V=800.0 PL=0
MOVL C02037 V=800.0 PL=0
MOVL C02038 V=800.0 PL=0
MOVL C02039 V=800.0 PL=0
MOVL C02040 V=800.0 PL=0
MOVL C02041 V=800.0 PL=0
MOVL C02042 V=800.0 PL=0
MOVL C02043 V=800.0 PL=0
MOVL C02044 V=800.0 PL=0
MOVL C02045 V=800.0 PL=0
MOVL C02046 V=800.0 PL=0
MOVL C02047 V=800.0 PL=0
MOVL C02048 V=800.0 PL=0
MOVL C02049 V=800.0 PL=0
MOVL C02050 V=800.0 PL=0
MOVL C02051 V=800.0 PL=0
MOVL C02052 V=800.0 PL=0
MOVL C02053 V=800.0 PL=0
MOVL C02054 V=800.0 PL=0
MOVL C02055 V=800.0 PL=0
MOVL C02056 V=800.0 PL=0
MOVL C02057 V=800.0 PL=0
MOVL C02058 V=800.0 PL=0
MOVL C02059 V=800.0 PL=0
MOVL C02060 V=800.0 PL=0
MOVL C02061 V=800.0 PL=0
MOVL C02062 V=800.0 PL=0
MOVL C02063 V=800.0 PL=0
MOVL C02064 V=800.0 PL=0
MOVL C02065 V=800.0 PL=0
MOVL C02066 V=800.0 PL=0
MOVL C02067 V=800.0 PL=0
MOVL C02068 V=800.0 PL=0
MOVL C02069 V=800.0 PL=0
MOVL C02070 V=800.0 PL=0
MOVL C02071 V=800.0 PL=0
MOVL C02072 V=800.0 PL=0
MOVL C02073 V=800.0 PL=0
MOVL C02074 V=800.0 PL=0
MOVL C02075 V=800.0 PL=0
MOVL C02076 V=800.0 PL=0
MOVL C02077 V=800.0 PL=0
MOVL C02078 V=800.0 PL=0
MOVL C02079 V=800.0 PL=0
MOVL C02080 V=800.0 PL=0
MOVL C02081 V=800.0 PL=0
MOVL C02082 V=800.0 PL=0
MOVL C02083 V=800.0 PL=0
MOVL C02084 V=800.0 PL=0
MOVL C02085 V=800.0 PL=0
MOVL C02086 V=800.0 PL=0
MOVL C02087 V=800.0 PL=0
MOVL C02088 V=800.0 PL=0
MOVL C02089 V=800.0 PL=0
MOVL C02090 V=800.0 PL=0
MOVL C02091 V=800.0 PL=0
MOVL C02092 V=800.0 PL=0
MOVL C02093 V=800.0 PL=0
MOVL C02094 V=800.0 PL=0
MOVL C02095 V=800.0 PL=0
MOVL C02096 V=800.0 PL=0
MOVL C02097 V=800.0 PL=0
MOVL C02098 V=800.0 PL=0
MOVL C02099 V=800.0 PL=0
MOVL C02100 V=800.0 PL=0
MOVL C02101 V=800.0 PL=0
MOVL C02102 V=800.0 PL=0
MOVL C02103 V=800.0 PL=0
MOVL C02104 V=800.0 PL=0
MOVL C02105 V=800.0 PL=0
MOVL C02106 V=800.0 PL=0
MOVL C02107 V=800.0 PL=0
MOVL C02108 V=800.0 PL=0
MOVL C02109 V=800.0 PL=0
MOVL C02110 V=800.0 PL=0
MOVL C02111 V=800.0 PL=0
MOVL C02112 V=800.0 PL=0
MOVL C02113 V=800.0 PL=0
MOVL C02114 V=800.0 PL=0
MOVL C02115 V=800.0 PL=0
MOVL C02116 V=800.0 PL=0
MOVL C02117 V=800.0 PL=0
MOVL C02118 V=800.0 PL=0
MOVL C02119 V=800.0 PL=0
MOVL C02120 V=800.0 PL=0
MOVL C02121 V=800.0 PL=0
MOVL C02122 V=800.0 PL=0
MOVL C02123 V=800.0 PL=0
MOVL C02124 V=800.0 PL=0
MOVL C02125 V=800.0 PL=0
MOVL C02126 V=800.0 PL=0
MOVL C02127 V=800.0 PL=0
MOVL C02128 V=800.0 PL=0
MOVL C02129 V=800.0 PL=0
MOVL C02130 V=800.0 PL=0
MOVL C02131 V=800.0 PL=0
MOVL C02132 V=800.0 PL=0
MOVL C02133 V=800.0 PL=0
MOVL C02134 V=800.0 PL=0
MOVL C02135 V=800.0 PL=0
MOVL C02136 V=800.0 PL=0
MOVL C02137 V=800.0 PL=0
MOVL C02138 V=800.0 PL=0
MOVL C02139 V=800.0 PL=0
MOVL C02140 V=800.0 PL=0
